  MoveL 5419 to (-31.64, 163.21, 88.06) mm, rotated rx 180 ry 0 rz 180 deg; joints [-52.884, -13.901, 88.099, 78.356, 54.505, -70.46]
  Call Extruder(2.18198)
  MoveL 5420 to (-31.93, 163.09, 88.06) mm, rotated rx 180 ry 0 rz -180 deg; joints [-52.91, -13.939, 88.128, 78.36, 54.532, -70.455]
  MoveL 5421 to (-31.93, 163.09, 88.06) mm, rotated rx 180 ry 0 rz -180 deg; joints [-52.91, -13.939, 88.128, 78.36, 54.532, -70.455]
  Call Extruder(2.36471)
  MoveL 5422 to (-32.22, 162.97, 88.06) mm, rotated rx 180 ry 0 rz 180 deg; joints [-52.936, -13.978, 88.158, 78.364, 54.558, -70.45]
  MoveL 5423 to (-32.22, 162.97, 88.06) mm, rotated rx 180 ry 0 rz 180 deg; joints [-52.936, -13.978, 88.158, 78.364, 54.558, -70.45]
  Call Extruder(2.53513)
  MoveL 5424 to (-32.49, 162.85, 88.06) mm, rotated rx -180 ry 0 rz 180 deg; joints [-52.96, -14.014, 88.185, 78.368, 54.583, -70.445]
  MoveL 5425 to (-32.49, 162.85, 88.06) mm, rotated rx -180 ry 0 rz 180 deg; joints [-52.96, -14.014, 88.185, 78.368, 54.583, -70.445]
  Call Extruder(2.69310)
  MoveL 5426 to (-32.74, 162.74, 88.06) mm, rotated rx 180 ry 0 rz 180 deg; joints [-52.982, -14.048, 88.211, 78.372, 54.605, -70.44]
  MoveL 5427 to (-32.74, 162.74, 88.06) mm, rotated rx 180 ry 0 rz 180 deg; joints [-52.982, -14.048, 88.211, 78.372, 54.605, -70.44]
  Call Extruder(2.85168)
  MoveL 5428 to (-32.99, 162.64, 88.06) mm, rotated rx 180 ry 0 rz -180 deg; joints [-53.004, -14.082, 88.236, 78.375, 54.627, -70.436]
  MoveL 5429 to (-32.99, 162.64, 88.06) mm, rotated rx 180 ry 0 rz -180 deg; joints [-53.004, -14.082, 88.236, 78.375, 54.627, -70.436]
  Call Extruder(3.05785)
  MoveL 5430 to (-33.29, 162.46, 88.06) mm, rotated rx 180 ry 0 rz 180 deg; joints [-53.026, -14.128, 88.271, 78.376, 54.651, -70.428]
  MoveL 5431 to (-33.29, 162.46, 88.06) mm, rotated rx 180 ry 0 rz 180 deg; joints [-53.026, -14.128, 88.271, 78.376, 54.651, -70.428]
  Call Extruder(3.26479)
  MoveL 5432 to (-33.6, 162.29, 88.06) mm, rotated rx 180 ry 0 rz 180 deg; joints [-53.049, -14.174, 88.306, 78.378, 54.674, -70.42]
  MoveL 5433 to (-33.6, 162.29, 88.06) mm, rotated rx 180 ry 0 rz 180 deg; joints [-53.049, -14.174, 88.306, 78.378, 54.674, -70.42]
  Call Extruder(3.47251)
  MoveL 5434 to (-33.9, 162.11, 88.06) mm, rotated rx 180 ry 0 rz 180 deg; joints [-53.071, -14.22, 88.34, 78.379, 54.698, -70.411]
  MoveL 5435 to (-33.9, 162.11, 88.06) mm, rotated rx 180 ry 0 rz 180 deg; joints [-53.071, -14.22, 88.34, 78.379, 54.698, -70.411]
  Call Extruder(3.68102)
  MoveL 5436 to (-34.21, 161.94, 88.06) mm, rotated rx 180 ry 0 rz 180 deg; joints [-53.094, -14.266, 88.375, 78.381, 54.721, -70.403]
  MoveL 5437 to (-34.21, 161.94, 88.06) mm, rotated rx 180 ry 0 rz 180 deg; joints [-53.094, -14.266, 88.375, 78.381, 54.721, -70.403]
  Call Extruder(3.86055)
  MoveL 5438 to (-34.45, 161.76, 88.06) mm, rotated rx 180 ry 0 rz 180 deg; joints [-53.109, -14.307, 88.406, 78.38, 54.737, -70.394]
  MoveL 5439 to (-34.45, 161.76, 88.06) mm, rotated rx 180 ry 0 rz 180 deg; joints [-53.109, -14.307, 88.406, 78.38, 54.737, -70.394]
  Call Extruder(4.19399)
  MoveL 5440 to (-34.9, 161.43, 88.06) mm, rotated rx 180 ry 0 rz 180 deg; joints [-53.135, -14.383, 88.463, 78.378, 54.766, -70.378]
  MoveL 5441 to (-34.9, 161.43, 88.06) mm, rotated rx 180 ry 0 rz 180 deg; joints [-53.135, -14.383, 88.463, 78.378, 54.766, -70.378]
  Call Extruder(4.52861)
  MoveL 5442 to (-35.35, 161.1, 88.06) mm, rotated rx -180 ry 0 rz 180 deg; joints [-53.163, -14.458, 88.52, 78.376, 54.795, -70.362]
  Call Extruder(5.35652)
  MoveL 5443 to (-36.39, 160.19, 88.06) mm, rotated rx 180 ry 0 rz 180 deg; joints [-53.209, -14.651, 88.664, 78.362, 54.849, -70.315]
  Call Extruder(6.18445)
  MoveL 5444 to (-37.3, 159.15, 88.06) mm, rotated rx 180 ry 0 rz -180 deg; joints [-53.227, -14.846, 88.809, 78.335, 54.876, -70.26]
  Call Extruder(6.35176)
  MoveL 5445 to (-37.47, 158.93, 88.06) mm, rotated rx 180 ry 0 rz -180 deg; joints [-53.227, -14.886, 88.839, 78.327, 54.878, -70.247]
  MoveL 5446 to (-37.47, 158.93, 88.06) mm, rotated rx 180 ry 0 rz -180 deg; joints [-53.227, -14.886, 88.839, 78.327, 54.878, -70.247]
  Call Extruder(6.68519)
  MoveL 5447 to (-37.8, 158.48, 88.06) mm, rotated rx -180 ry 0 rz 180 deg; joints [-53.226, -14.965, 88.897, 78.313, 54.881, -70.223]
  MoveL 5448 to (-37.8, 158.48, 88.06) mm, rotated rx -180 ry 0 rz 180 deg; joints [-53.226, -14.965, 88.897, 78.313, 54.881, -70.223]
  Call Extruder(7.01743)
  MoveL 5449 to (-38.12, 158.02, 88.06) mm, rotated rx -180 ry 0 rz 180 deg; joints [-53.224, -15.044, 88.956, 78.298, 54.884, -70.198]
  MoveL 5450 to (-38.12, 158.02, 88.06) mm, rotated rx -180 ry 0 rz 180 deg; joints [-53.224, -15.044, 88.956, 78.298, 54.884, -70.198]
  Call Extruder(7.13510)
  MoveL 5451 to (-38.22, 157.85, 88.06) mm, rotated rx 180 ry 0 rz 180 deg; joints [-53.221, -15.072, 88.977, 78.292, 54.882, -70.188]
  MoveL 5452 to (-38.22, 157.85, 88.06) mm, rotated rx 180 ry 0 rz 180 deg; joints [-53.221, -15.072, 88.977, 78.292, 54.882, -70.188]
  Call Extruder(7.34283)
  MoveL 5453 to (-38.4, 157.55, 88.06) mm, rotated rx -180 ry 0 rz 180 deg; joints [-53.214, -15.121, 89.013, 78.28, 54.878, -70.171]
  MoveL 5454 to (-38.4, 157.55, 88.06) mm, rotated rx -180 ry 0 rz 180 deg; joints [-53.214, -15.121, 89.013, 78.28, 54.878, -70.171]
  Call Extruder(7.54978)
  MoveL 5455 to (-38.57, 157.25, 88.06) mm, rotated rx 180 ry 0 rz 180 deg; joints [-53.207, -15.171, 89.05, 78.268, 54.874, -70.154]
  MoveL 5456 to (-38.57, 157.25, 88.06) mm, rotated rx 180 ry 0 rz 180 deg; joints [-53.207, -15.171, 89.05, 78.268, 54.874, -70.154]
  Call Extruder(7.75595)
  MoveL 5457 to (-38.75, 156.94, 88.06) mm, rotated rx -180 ry 0 rz 180 deg; joints [-53.2, -15.22, 89.086, 78.256, 54.87, -70.137]
  MoveL 5458 to (-38.75, 156.94, 88.06) mm, rotated rx -180 ry 0 rz 180 deg; joints [-53.2, -15.22, 89.086, 78.256, 54.87, -70.137]
  Call Extruder(7.93763)
  MoveL 5459 to (-38.89, 156.66, 88.06) mm, rotated rx -180 ry 0 rz 180 deg; joints [-53.191, -15.263, 89.118, 78.245, 54.864, -70.121]
  MoveL 5460 to (-38.89, 156.66, 88.06) mm, rotated rx -180 ry 0 rz 180 deg; joints [-53.191, -15.263, 89.118, 78.245, 54.864, -70.121]
  Call Extruder(8.09561)
  MoveL 5461 to (-39, 156.42, 88.06) mm, rotated rx -180 ry 0 rz 180 deg; joints [-53.18, -15.301, 89.145, 78.234, 54.856, -70.107]
  MoveL 5462 to (-39, 156.42, 88.06) mm, rotated rx -180 ry 0 rz 180 deg; joints [-53.18, -15.301, 89.145, 78.234, 54.856, -70.107]
  Call Extruder(8.25300)
  MoveL 5463 to (-39.11, 156.17, 88.06) mm, rotated rx -180 ry 0 rz 180 deg; joints [-53.17, -15.338, 89.173, 78.222, 54.848, -70.092]
  MoveL 5464 to (-39.11, 156.17, 88.06) mm, rotated rx -180 ry 0 rz 180 deg; joints [-53.17, -15.338, 89.173, 78.222, 54.848, -70.092]
  Call Extruder(8.43571)
  MoveL 5465 to (-39.22, 155.88, 88.06) mm, rotated rx 180 ry 0 rz 180 deg; joints [-53.156, -15.381, 89.205, 78.209, 54.838, -70.075]
  MoveL 5466 to (-39.22, 155.88, 88.06) mm, rotated rx 180 ry 0 rz 180 deg; joints [-53.156, -15.381, 89.205, 78.209, 54.838, -70.075]
  Call Extruder(8.61768)
  MoveL 5467 to (-39.35, 155.58, 88.06) mm, rotated rx 180 ry 0 rz 180 deg; joints [-53.143, -15.425, 89.236, 78.195, 54.828, -70.058]
  MoveL 5468 to (-39.35, 155.58, 88.06) mm, rotated rx 180 ry 0 rz 180 deg; joints [-53.143, -15.425, 89.236, 78.195, 54.828, -70.058]
  Call Extruder(8.76501)
  MoveL 5469 to (-39.44, 155.34, 88.06) mm, rotated rx 180 ry 0 rz 180 deg; joints [-53.131, -15.459, 89.262, 78.184, 54.819, -70.044]
  MoveL 5470 to (-39.44, 155.34, 88.06) mm, rotated rx 180 ry 0 rz 180 deg; joints [-53.131, -15.459, 89.262, 78.184, 54.819, -70.044]
  Call Extruder(8.87824)
  MoveL 5471 to (-39.5, 155.15, 88.06) mm, rotated rx -180 ry 0 rz 180 deg; joints [-53.121, -15.486, 89.281, 78.175, 54.81, -70.033]
  MoveL 5472 to (-39.5, 155.15, 88.06) mm, rotated rx -180 ry 0 rz 180 deg; joints [-53.121, -15.486, 89.281, 78.175, 54.81, -70.033]
  Call Extruder(8.99103)
  MoveL 5473 to (-39.56, 154.97, 88.06) mm, rotated rx 180 ry 0 rz 180 deg; joints [-53.11, -15.513, 89.301, 78.165, 54.801, -70.022]
  MoveL 5474 to (-39.56, 154.97, 88.06) mm, rotated rx 180 ry 0 rz 180 deg; joints [-53.11, -15.513, 89.301, 78.165, 54.801, -70.022]
  Call Extruder(9.10338)
  MoveL 5475 to (-39.62, 154.78, 88.06) mm, rotated rx 180 ry 0 rz 180 deg; joints [-53.099, -15.539, 89.32, 78.156, 54.793, -70.011]
  MoveL 5476 to (-39.62, 154.78, 88.06) mm, rotated rx 180 ry 0 rz 180 deg; joints [-53.099, -15.539, 89.32, 78.156, 54.793, -70.011]
  Call Extruder(9.21528)
  MoveL 5477 to (-39.68, 154.59, 88.06) mm, rotated rx 180 ry 0 rz 180 deg; joints [-53.088, -15.566, 89.34, 78.146, 54.784, -70]
  MoveL 5478 to (-39.68, 154.59, 88.06) mm, rotated rx 180 ry 0 rz 180 deg; joints [-53.088, -15.566, 89.34, 78.146, 54.784, -70]
  Call Extruder(9.33668)
  MoveL 5479 to (-39.75, 154.38, 88.06) mm, rotated rx -180 ry 0 rz 180 deg; joints [-53.076, -15.594, 89.361, 78.136, 54.774, -69.988]
  MoveL 5480 to (-39.75, 154.38, 88.06) mm, rotated rx -180 ry 0 rz 180 deg; joints [-53.076, -15.594, 89.361, 78.136, 54.774, -69.988]
  Call Extruder(9.46747)
  MoveL 5481 to (-39.81, 154.16, 88.06) mm, rotated rx 180 ry 0 rz 180 deg; joints [-53.063, -15.625, 89.383, 78.124, 54.763, -69.974]
  MoveL 5482 to (-39.81, 154.16, 88.06) mm, rotated rx 180 ry 0 rz 180 deg; joints [-53.063, -15.625, 89.383, 78.124, 54.763, -69.974]
  Call Extruder(9.59770)
  MoveL 5483 to (-39.88, 153.94, 88.06) mm, rotated rx 180 ry 0 rz 180 deg; joints [-53.049, -15.656, 89.406, 78.113, 54.752, -69.961]
  MoveL 5484 to (-39.88, 153.94, 88.06) mm, rotated rx 180 ry 0 rz 180 deg; joints [-53.049, -15.656, 89.406, 78.113, 54.752, -69.961]
  Call Extruder(9.72737)
  MoveL 5485 to (-39.95, 153.71, 88.06) mm, rotated rx 180 ry 0 rz 180 deg; joints [-53.036, -15.687, 89.428, 78.102, 54.741, -69.948]
  MoveL 5486 to (-39.95, 153.71, 88.06) mm, rotated rx 180 ry 0 rz 180 deg; joints [-53.036, -15.687, 89.428, 78.102, 54.741, -69.948]
  Call Extruder(9.85647)
  MoveL 5487 to (-40.02, 153.49, 88.06) mm, rotated rx 180 ry 0 rz 180 deg; joints [-53.022, -15.718, 89.451, 78.09, 54.73, -69.934]
  MoveL 5488 to (-40.02, 153.49, 88.06) mm, rotated rx 180 ry 0 rz 180 deg; joints [-53.022, -15.718, 89.451, 78.09, 54.73, -69.934]
  Call Extruder(9.97156)
  MoveL 5489 to (-40.06, 153.28, 88.06) mm, rotated rx -180 ry 0 rz 180 deg; joints [-53.007, -15.745, 89.471, 78.079, 54.718, -69.922]
  MoveL 5490 to (-40.06, 153.28, 88.06) mm, rotated rx -180 ry 0 rz 180 deg; joints [-53.007, -15.745, 89.471, 78.079, 54.718, -69.922]
  Call Extruder(10.08619)
  MoveL 5491 to (-40.11, 153.08, 88.06) mm, rotated rx 180 ry 0 rz 180 deg; joints [-52.993, -15.772, 89.49, 78.067, 54.706, -69.91]
  MoveL 5492 to (-40.11, 153.08, 88.06) mm, rotated rx 180 ry 0 rz 180 deg; joints [-52.993, -15.772, 89.49, 78.067, 54.706, -69.91]
  Call Extruder(10.20038)
  MoveL 5493 to (-40.15, 152.88, 88.06) mm, rotated rx 180 ry 0 rz 180 deg; joints [-52.978, -15.799, 89.509, 78.056, 54.693, -69.897]
  MoveL 5494 to (-40.15, 152.88, 88.06) mm, rotated rx 180 ry 0 rz 180 deg; joints [-52.978, -15.799, 89.509, 78.056, 54.693, -69.897]
  Call Extruder(10.31411)
  MoveL 5495 to (-40.2, 152.67, 88.06) mm, rotated rx 180 ry 0 rz 180 deg; joints [-52.963, -15.826, 89.529, 78.045, 54.681, -69.885]
  MoveL 5496 to (-40.2, 152.67, 88.06) mm, rotated rx 180 ry 0 rz 180 deg; joints [-52.963, -15.826, 89.529, 78.045, 54.681, -69.885]
  Call Extruder(10.43953)
  MoveL 5497 to (-40.24, 152.45, 88.06) mm, rotated rx 180 ry 0 rz 180 deg; joints [-52.946, -15.855, 89.55, 78.032, 54.667, -69.871]
  MoveL 5498 to (-40.24, 152.45, 88.06) mm, rotated rx 180 ry 0 rz 180 deg; joints [-52.946, -15.855, 89.55, 78.032, 54.667, -69.871]
  Call Extruder(10.57651)
  MoveL 5499 to (-40.29, 152.2, 88.06) mm, rotated rx 180 ry 0 rz 180 deg; joints [-52.928, -15.887, 89.574, 78.018, 54.651, -69.856]
  MoveL 5500 to (-40.29, 152.2, 88.06) mm, rotated rx 180 ry 0 rz 180 deg; joints [-52.928, -15.887, 89.574, 78.018, 54.651, -69.856]
  Call Extruder(10.71287)
  MoveL 5501 to (-40.34, 151.95, 88.06) mm, rotated rx -180 ry 0 rz 180 deg; joints [-52.909, -15.92, 89.597, 78.004, 54.635, -69.841]
  MoveL 5502 to (-40.34, 151.95, 88.06) mm, rotated rx -180 ry 0 rz 180 deg; joints [-52.909, -15.92, 89.597, 78.004, 54.635, -69.841]
  Call Extruder(10.84863)
  MoveL 5503 to (-40.39, 151.7, 88.06) mm, rotated rx 180 ry 0 rz -180 deg; joints [-52.89, -15.952, 89.621, 77.99, 54.62, -69.825]
  MoveL 5504 to (-40.39, 151.7, 88.06) mm, rotated rx 180 ry 0 rz -180 deg; joints [-52.89, -15.952, 89.621, 77.99, 54.62, -69.825]
  Call Extruder(10.98377)
  MoveL 5505 to (-40.44, 151.45, 88.06) mm, rotated rx 180 ry 0 rz -180 deg; joints [-52.871, -15.984, 89.644, 77.976, 54.604, -69.81]
  MoveL 5506 to (-40.44, 151.45, 88.06) mm, rotated rx 180 ry 0 rz -180 deg; joints [-52.871, -15.984, 89.644, 77.976, 54.604, -69.81]
  Call Extruder(11.11831)
  MoveL 5507 to (-40.49, 151.2, 88.06) mm, rotated rx -180 ry 0 rz 180 deg; joints [-52.853, -16.016, 89.667, 77.962, 54.588, -69.795]
  MoveL 5508 to (-40.49, 151.2, 88.06) mm, rotated rx -180 ry 0 rz 180 deg; joints [-52.853, -16.016, 89.667, 77.962, 54.588, -69.795]
  Call Extruder(11.25223)
  MoveL 5509 to (-40.54, 150.95, 88.06) mm, rotated rx -180 ry 0 rz 180 deg; joints [-52.834, -16.048, 89.69, 77.947, 54.572, -69.779]
  MoveL 5510 to (-40.54, 150.95, 88.06) mm, rotated rx -180 ry 0 rz 180 deg; joints [-52.834, -16.048, 89.69, 77.947, 54.572, -69.779]
  Call Extruder(11.40009)
  MoveL 5511 to (-40.59, 150.67, 88.06) mm, rotated rx 180 ry 0 rz 180 deg; joints [-52.812, -16.084, 89.716, 77.931, 54.554, -69.762]
  MoveL 5512 to (-40.59, 150.67, 88.06) mm, rotated rx 180 ry 0 rz 180 deg; joints [-52.812, -16.084, 89.716, 77.931, 54.554, -69.762]
  Call Extruder(11.56181)
  MoveL 5513 to (-40.64, 150.37, 88.06) mm, rotated rx 180 ry 0 rz 180 deg; joints [-52.787, -16.122, 89.744, 77.913, 54.533, -69.743]
  MoveL 5514 to (-40.64, 150.37, 88.06) mm, rotated rx 180 ry 0 rz 180 deg; joints [-52.787, -16.122, 89.744, 77.913, 54.533, -69.743]
  Call Extruder(11.72281)
  MoveL 5515 to (-40.69, 150.06, 88.06) mm, rotated rx 180 ry 0 rz 180 deg; joints [-52.762, -16.161, 89.771, 77.895, 54.512, -69.724]
  MoveL 5516 to (-40.69, 150.06, 88.06) mm, rotated rx 180 ry 0 rz 180 deg; joints [-52.762, -16.161, 89.771, 77.895, 54.512, -69.724]
  Call Extruder(11.88308)
  MoveL 5517 to (-40.73, 149.76, 88.06) mm, rotated rx 180 ry 0 rz 180 deg; joints [-52.737, -16.199, 89.799, 77.877, 54.491, -69.705]
  MoveL 5518 to (-40.73, 149.76, 88.06) mm, rotated rx 180 ry 0 rz 180 deg; joints [-52.737, -16.199, 89.799, 77.877, 54.491, -69.705]
  Call Extruder(12.04262)
  MoveL 5519 to (-40.78, 149.45, 88.06) mm, rotated rx -180 ry 0 rz -180 deg; joints [-52.712, -16.237, 89.827, 77.859, 54.469, -69.686]
  MoveL 5520 to (-40.78, 149.45, 88.06) mm, rotated rx -180 ry 0 rz -180 deg; joints [-52.712, -16.237, 89.827, 77.859, 54.469, -69.686]
  Call Extruder(12.20144)
  MoveL 5521 to (-40.83, 149.14, 88.06) mm, rotated rx -180 ry 0 rz -180 deg; joints [-52.687, -16.276, 89.854, 77.841, 54.448, -69.667]
  MoveL 5522 to (-40.83, 149.14, 88.06) mm, rotated rx -180 ry 0 rz -180 deg; joints [-52.687, -16.276, 89.854, 77.841, 54.448, -69.667]
  Call Extruder(12.38010)
  MoveL 5523 to (-40.88, 148.8, 88.06) mm, rotated rx 180 ry 0 rz 180 deg; joints [-52.658, -16.319, 89.885, 77.82, 54.423, -69.645]
  MoveL 5524 to (-40.88, 148.8, 88.06) mm, rotated rx 180 ry 0 rz 180 deg; joints [-52.658, -16.319, 89.885, 77.82, 54.423, -69.645]
  Call Extruder(12.57854)
  MoveL 5525 to (-40.93, 148.41, 88.06) mm, rotated rx 180 ry 0 rz 180 deg; joints [-52.624, -16.366, 89.919, 77.796, 54.394, -69.62]
  MoveL 5526 to (-40.93, 148.41, 88.06) mm, rotated rx 180 ry 0 rz 180 deg; joints [-52.624, -16.366, 89.919, 77.796, 54.394, -69.62]
  Call Extruder(12.77611)
  MoveL 5527 to (-40.97, 148.02, 88.06) mm, rotated rx 180 ry 0 rz 180 deg; joints [-52.59, -16.413, 89.953, 77.772, 54.365, -69.596]
  MoveL 5528 to (-40.97, 148.02, 88.06) mm, rotated rx 180 ry 0 rz 180 deg; joints [-52.59, -16.413, 89.953, 77.772, 54.365, -69.596]
  Call Extruder(12.97282)
  MoveL 5529 to (-41.02, 147.63, 88.06) mm, rotated rx 180 ry 0 rz 180 deg; joints [-52.556, -16.46, 89.986, 77.748, 54.336, -69.571]
  MoveL 5530 to (-41.02, 147.63, 88.06) mm, rotated rx 180 ry 0 rz 180 deg; joints [-52.556, -16.46, 89.986, 77.748, 54.336, -69.571]
  Call Extruder(13.16866)
  MoveL 5531 to (-41.06, 147.25, 88.06) mm, rotated rx 180 ry 0 rz 180 deg; joints [-52.521, -16.508, 90.02, 77.724, 54.307, -69.546]
  MoveL 5532 to (-41.06, 147.25, 88.06) mm, rotated rx 180 ry 0 rz 180 deg; joints [-52.521, -16.508, 90.02, 77.724, 54.307, -69.546]
  Call Extruder(13.46406)
  MoveL 5533 to (-41.11, 146.66, 88.06) mm, rotated rx 180 ry 0 rz 180 deg; joints [-52.466, -16.577, 90.07, 77.686, 54.259, -69.508]
  MoveL 5534 to (-41.11, 146.66, 88.06) mm, rotated rx 180 ry 0 rz 180 deg; joints [-52.466, -16.577, 90.07, 77.686, 54.259, -69.508]
  Call Extruder(13.75812)
  MoveL 5535 to (-41.15, 146.07, 88.06) mm, rotated rx -180 ry 0 rz 180 deg; joints [-52.411, -16.647, 90.119, 77.648, 54.212, -69.47]
  MoveL 5536 to (-41.15, 146.07, 88.06) mm, rotated rx -180 ry 0 rz 180 deg; joints [-52.411, -16.647, 90.119, 77.648, 54.212, -69.47]
  Call Extruder(14.05085)
  MoveL 5537 to (-41.2, 145.48, 88.06) mm, rotated rx -180 ry 0 rz 180 deg; joints [-52.355, -16.717, 90.169, 77.61, 54.164, -69.432]
  MoveL 5538 to (-41.2, 145.48, 88.06) mm, rotated rx -180 ry 0 rz 180 deg; joints [-52.355, -16.717, 90.169, 77.61, 54.164, -69.432]
  Call Extruder(14.62431)
  MoveL 5539 to (-41.25, 144.32, 88.06) mm, rotated rx 180 ry 0 rz 180 deg; joints [-52.239, -16.85, 90.263, 77.532, 54.063, -69.356]
  MoveL 5540 to (-41.25, 144.32, 88.06) mm, rotated rx 180 ry 0 rz 180 deg; joints [-52.239, -16.85, 90.263, 77.532, 54.063, -69.356]
  Call Extruder(15.33827)
  MoveL 5541 to (-41.29, 142.86, 88.06) mm, rotated rx 180 ry 0 rz 180 deg; joints [-52.09, -17.014, 90.38, 77.432, 53.934, -69.259]
  Call Extruder(57.40309)
  MoveL 5542 to (-41.29, 57.14, 88.06) mm, rotated rx 180 ry 0 rz 180 deg; joints [-40.759, -25.558, 95.751, 68.538, 44.549, -61.117]
  Call Extruder(57.83165)
  MoveL 5543 to (-41.27, 56.26, 88.06) mm, rotated rx -180 ry 0 rz -180 deg; joints [-40.614, -25.632, 95.792, 68.407, 44.435, -61.001]
  MoveL 5544 to (-41.27, 56.26, 88.06) mm, rotated rx -180 ry 0 rz -180 deg; joints [-40.614, -25.632, 95.792, 68.407, 44.435, -61.001]
  Call Extruder(58.40510)
  MoveL 5545 to (-41.23, 55.1, 88.06) mm, rotated rx 180 ry 0 rz -180 deg; joints [-40.419, -25.728, 95.844, 68.23, 44.28, -60.846]
  MoveL 5546 to (-41.23, 55.1, 88.06) mm, rotated rx 180 ry 0 rz -180 deg; joints [-40.419, -25.728, 95.844, 68.23, 44.28, -60.846]
  Call Extruder(58.83942)
  MoveL 5547 to (-41.18, 54.23, 88.06) mm, rotated rx 180 ry 0 rz 180 deg; joints [-40.269, -25.799, 95.883, 68.094, 44.161, -60.728]
  MoveL 5548 to (-41.18, 54.23, 88.06) mm, rotated rx 180 ry 0 rz 180 deg; joints [-40.269, -25.799, 95.883, 68.094, 44.161, -60.728]
  Call Extruder(59.13348)
  MoveL 5549 to (-41.13, 53.64, 88.06) mm, rotated rx 180 ry 0 rz 180 deg; joints [-40.165, -25.845, 95.908, 68.001, 44.078, -60.648]
  MoveL 5550 to (-41.13, 53.64, 88.06) mm, rotated rx 180 ry 0 rz 180 deg; joints [-40.165, -25.845, 95.908, 68.001, 44.078, -60.648]
  Call Extruder(59.42888)
  MoveL 5551 to (-41.09, 53.05, 88.06) mm, rotated rx 180 ry 0 rz 180 deg; joints [-40.062, -25.891, 95.933, 67.908, 43.996, -60.568]
  MoveL 5552 to (-41.09, 53.05, 88.06) mm, rotated rx 180 ry 0 rz 180 deg; joints [-40.062, -25.891, 95.933, 67.908, 43.996, -60.568]
  Call Extruder(59.67512)
  MoveL 5553 to (-41.04, 52.56, 88.06) mm, rotated rx 180 ry 0 rz 180 deg; joints [-39.975, -25.928, 95.953, 67.83, 43.927, -60.501]
  MoveL 5554 to (-41.04, 52.56, 88.06) mm, rotated rx 180 ry 0 rz 180 deg; joints [-39.975, -25.928, 95.953, 67.83, 43.927, -60.501]
  Call Extruder(59.87182)
  MoveL 5555 to (-40.99, 52.17, 88.06) mm, rotated rx -180 ry 0 rz 180 deg; joints [-39.904, -25.957, 95.969, 67.768, 43.87, -60.447]
  MoveL 5556 to (-40.99, 52.17, 88.06) mm, rotated rx -180 ry 0 rz 180 deg; joints [-39.904, -25.957, 95.969, 67.768, 43.87, -60.447]
  Call Extruder(60.06940)
  MoveL 5557 to (-40.95, 51.78, 88.06) mm, rotated rx 180 ry 0 rz 180 deg; joints [-39.833, -25.985, 95.984, 67.705, 43.814, -60.394]
  MoveL 5558 to (-40.95, 51.78, 88.06) mm, rotated rx 180 ry 0 rz 180 deg; joints [-39.833, -25.985, 95.984, 67.705, 43.814, -60.394]
  Call Extruder(60.26784)
  MoveL 5559 to (-40.9, 51.4, 88.06) mm, rotated rx -180 ry 0 rz -180 deg; joints [-39.763, -26.013, 96, 67.642, 43.757, -60.34]
  MoveL 5560 to (-40.9, 51.4, 88.06) mm, rotated rx -180 ry 0 rz -180 deg; joints [-39.763, -26.013, 96, 67.642, 43.757, -60.34]
  Call Extruder(60.46715)
  MoveL 5561 to (-40.86, 51.01, 88.06) mm, rotated rx 180 ry 0 rz 180 deg; joints [-39.692, -26.042, 96.015, 67.578, 43.7, -60.286]
  MoveL 5562 to (-40.86, 51.01, 88.06) mm, rotated rx 180 ry 0 rz 180 deg; joints [-39.692, -26.042, 96.015, 67.578, 43.7, -60.286]
  Call Extruder(60.62596)
  MoveL 5563 to (-40.81, 50.7, 88.06) mm, rotated rx -180 ry 0 rz -180 deg; joints [-39.634, -26.063, 96.026, 67.528, 43.654, -60.243]
  MoveL 5564 to (-40.81, 50.7, 88.06) mm, rotated rx -180 ry 0 rz -180 deg; joints [-39.634, -26.063, 96.026, 67.528, 43.654, -60.243]
  Call Extruder(60.78551)
  MoveL 5565 to (-40.76, 50.4, 88.06) mm, rotated rx 180 ry 0 rz -180 deg; joints [-39.576, -26.084, 96.038, 67.477, 43.607, -60.2]
  MoveL 5566 to (-40.76, 50.4, 88.06) mm, rotated rx 180 ry 0 rz -180 deg; joints [-39.576, -26.084, 96.038, 67.477, 43.607, -60.2]
  Call Extruder(60.94578)
  MoveL 5567 to (-40.71, 50.09, 88.06) mm, rotated rx 180 ry 0 rz -180 deg; joints [-39.518, -26.104, 96.049, 67.426, 43.561, -60.157]
  MoveL 5568 to (-40.71, 50.09, 88.06) mm, rotated rx 180 ry 0 rz -180 deg; joints [-39.518, -26.104, 96.049, 67.426, 43.561, -60.157]
  Call Extruder(61.10677)
  MoveL 5569 to (-40.66, 49.79, 88.06) mm, rotated rx 180 ry 0 rz 180 deg; joints [-39.46, -26.125, 96.06, 67.374, 43.514, -60.114]
  MoveL 5570 to (-40.66, 49.79, 88.06) mm, rotated rx 180 ry 0 rz 180 deg; joints [-39.46, -26.125, 96.06, 67.374, 43.514, -60.114]
  Call Extruder(61.26850)
  MoveL 5571 to (-40.61, 49.48, 88.06) mm, rotated rx -180 ry 0 rz 180 deg; joints [-39.402, -26.146, 96.072, 67.323, 43.468, -60.07]
  MoveL 5572 to (-40.61, 49.48, 88.06) mm, rotated rx -180 ry 0 rz 180 deg; joints [-39.402, -26.146, 96.072, 67.323, 43.468, -60.07]
  Call Extruder(61.43095)
  MoveL 5573 to (-40.57, 49.17, 88.06) mm, rotated rx 180 ry 0 rz 180 deg; joints [-39.344, -26.167, 96.083, 67.272, 43.421, -60.027]
  MoveL 5574 to (-40.57, 49.17, 88.06) mm, rotated rx 180 ry 0 rz 180 deg; joints [-39.344, -26.167, 96.083, 67.272, 43.421, -60.027]
  Call Extruder(61.56488)
  MoveL 5575 to (-40.52, 48.93, 88.06) mm, rotated rx 180 ry 0 rz 180 deg; joints [-39.296, -26.183, 96.092, 67.229, 43.382, -59.991]
  MoveL 5576 to (-40.52, 48.93, 88.06) mm, rotated rx 180 ry 0 rz 180 deg; joints [-39.296, -26.183, 96.092, 67.229, 43.382, -59.991]
  Call Extruder(61.69941)
  MoveL 5577 to (-40.47, 48.68, 88.06) mm, rotated rx -180 ry 0 rz 180 deg; joints [-39.247, -26.199, 96.1, 67.186, 43.342, -59.955]
  MoveL 5578 to (-40.47, 48.68, 88.06) mm, rotated rx -180 ry 0 rz 180 deg; joints [-39.247, -26.199, 96.1, 67.186, 43.342, -59.955]
  Call Extruder(61.83456)
  MoveL 5579 to (-40.42, 48.43, 88.06) mm, rotated rx 180 ry 0 rz 180 deg; joints [-39.198, -26.215, 96.109, 67.143, 43.303, -59.92]
  MoveL 5580 to (-40.42, 48.43, 88.06) mm, rotated rx 180 ry 0 rz 180 deg; joints [-39.198, -26.215, 96.109, 67.143, 43.303, -59.92]
  Call Extruder(61.97031)
  MoveL 5581 to (-40.37, 48.18, 88.06) mm, rotated rx -180 ry 0 rz 180 deg; joints [-39.149, -26.231, 96.117, 67.101, 43.263, -59.884]
  MoveL 5582 to (-40.37, 48.18, 88.06) mm, rotated rx -180 ry 0 rz 180 deg; joints [-39.149, -26.231, 96.117, 67.101, 43.263, -59.884]
  Call Extruder(62.10668)
  MoveL 5583 to (-40.32, 47.93, 88.06) mm, rotated rx -180 ry 0 rz 180 deg; joints [-39.1, -26.246, 96.126, 67.058, 43.224, -59.848]
  MoveL 5584 to (-40.32, 47.93, 88.06) mm, rotated rx -180 ry 0 rz 180 deg; joints [-39.1, -26.246, 96.126, 67.058, 43.224, -59.848]
  Call Extruder(62.24365)
  MoveL 5585 to (-40.27, 47.68, 88.06) mm, rotated rx 180 ry 0 rz 180 deg; joints [-39.051, -26.262, 96.134, 67.015, 43.185, -59.812]
  MoveL 5586 to (-40.27, 47.68, 88.06) mm, rotated rx 180 ry 0 rz 180 deg; joints [-39.051, -26.262, 96.134, 67.015, 43.185, -59.812]
  Call Extruder(62.38124)
  MoveL 5587 to (-40.22, 47.43, 88.06) mm, rotated rx 180 ry 0 rz 180 deg; joints [-39.002, -26.278, 96.142, 66.971, 43.145, -59.776]
  MoveL 5588 to (-40.22, 47.43, 88.06) mm, rotated rx 180 ry 0 rz 180 deg; joints [-39.002, -26.278, 96.142, 66.971, 43.145, -59.776]
  Call Extruder(62.49497)
  MoveL 5589 to (-40.17, 47.23, 88.06) mm, rotated rx -180 ry 0 rz 180 deg; joints [-38.962, -26.29, 96.149, 66.936, 43.112, -59.746]
  MoveL 5590 to (-40.17, 47.23, 88.06) mm, rotated rx -180 ry 0 rz 180 deg; joints [-38.962, -26.29, 96.149, 66.936, 43.112, -59.746]
  Call Extruder(62.60915)
  MoveL 5591 to (-40.13, 47.02, 88.06) mm, rotated rx -180 ry 0 rz 180 deg; joints [-38.921, -26.303, 96.156, 66.9, 43.079, -59.716]
  MoveL 5592 to (-40.13, 47.02, 88.06) mm, rotated rx -180 ry 0 rz 180 deg; joints [-38.921, -26.303, 96.156, 66.9, 43.079, -59.716]
  Call Extruder(62.72378)
  MoveL 5593 to (-40.08, 46.82, 88.06) mm, rotated rx -180 ry 0 rz 180 deg; joints [-38.88, -26.315, 96.163, 66.864, 43.046, -59.687]
  MoveL 5594 to (-40.08, 46.82, 88.06) mm, rotated rx -180 ry 0 rz 180 deg; joints [-38.88, -26.315, 96.163, 66.864, 43.046, -59.687]
  Call Extruder(62.83887)
  MoveL 5595 to (-40.04, 46.61, 88.06) mm, rotated rx -180 ry 0 rz 180 deg; joints [-38.839, -26.328, 96.169, 66.828, 43.013, -59.657]
  MoveL 5596 to (-40.04, 46.61, 88.06) mm, rotated rx -180 ry 0 rz 180 deg; joints [-38.839, -26.328, 96.169, 66.828, 43.013, -59.657]
  Call Extruder(62.96111)
  MoveL 5597 to (-39.98, 46.4, 88.06) mm, rotated rx 180 ry 0 rz 180 deg; joints [-38.795, -26.34, 96.176, 66.79, 42.977, -59.625]
  MoveL 5598 to (-39.98, 46.4, 88.06) mm, rotated rx 180 ry 0 rz 180 deg; joints [-38.795, -26.34, 96.176, 66.79, 42.977, -59.625]
  Call Extruder(63.09077)
  MoveL 5599 to (-39.92, 46.18, 88.06) mm, rotated rx 180 ry 0 rz 180 deg; joints [-38.748, -26.351, 96.182, 66.75, 42.938, -59.592]
  MoveL 5600 to (-39.92, 46.18, 88.06) mm, rotated rx 180 ry 0 rz 180 deg; joints [-38.748, -26.351, 96.182, 66.75, 42.938, -59.592]
  Call Extruder(63.22100)
  MoveL 5601 to (-39.85, 45.95, 88.06) mm, rotated rx 180 ry 0 rz 180 deg; joints [-38.7, -26.363, 96.188, 66.709, 42.9, -59.559]
  MoveL 5602 to (-39.85, 45.95, 88.06) mm, rotated rx 180 ry 0 rz 180 deg; joints [-38.7, -26.363, 96.188, 66.709, 42.9, -59.559]
  Call Extruder(63.35179)
  MoveL 5603 to (-39.78, 45.73, 88.06) mm, rotated rx 180 ry 0 rz 180 deg; joints [-38.653, -26.374, 96.194, 66.668, 42.861, -59.526]
  MoveL 5604 to (-39.78, 45.73, 88.06) mm, rotated rx 180 ry 0 rz 180 deg; joints [-38.653, -26.374, 96.194, 66.668, 42.861, -59.526]
  Call Extruder(63.48315)
  MoveL 5605 to (-39.71, 45.51, 88.06) mm, rotated rx -180 ry 0 rz 180 deg; joints [-38.605, -26.386, 96.2, 66.628, 42.822, -59.493]
  MoveL 5606 to (-39.71, 45.51, 88.06) mm, rotated rx -180 ry 0 rz 180 deg; joints [-38.605, -26.386, 96.2, 66.628, 42.822, -59.493]
  Call Extruder(63.59505)
  MoveL 5607 to (-39.65, 45.32, 88.06) mm, rotated rx 180 ry 0 rz 180 deg; joints [-38.565, -26.395, 96.205, 66.593, 42.789, -59.465]
  MoveL 5608 to (-39.65, 45.32, 88.06) mm, rotated rx 180 ry 0 rz 180 deg; joints [-38.565, -26.395, 96.205, 66.593, 42.789, -59.465]
  Call Extruder(63.70740)
  MoveL 5609 to (-39.59, 45.13, 88.06) mm, rotated rx 180 ry 0 rz 180 deg; joints [-38.524, -26.404, 96.21, 66.558, 42.756, -59.437]
  MoveL 5610 to (-39.59, 45.13, 88.06) mm, rotated rx 180 ry 0 rz 180 deg; joints [-38.524, -26.404, 96.21, 66.558, 42.756, -59.437]
  Call Extruder(63.82019)
  MoveL 5611 to (-39.53, 44.94, 88.06) mm, rotated rx 180 ry 0 rz 180 deg; joints [-38.483, -26.414, 96.215, 66.524, 42.722, -59.409]
  MoveL 5612 to (-39.53, 44.94, 88.06) mm, rotated rx 180 ry 0 rz 180 deg; joints [-38.483, -26.414, 96.215, 66.524, 42.722, -59.409]
  Call Extruder(63.93342)
  MoveL 5613 to (-39.47, 44.75, 88.06) mm, rotated rx 180 ry 0 rz 180 deg; joints [-38.443, -26.423, 96.22, 66.489, 42.689, -59.38]
  MoveL 5614 to (-39.47, 44.75, 88.06) mm, rotated rx 180 ry 0 rz 180 deg; joints [-38.443, -26.423, 96.22, 66.489, 42.689, -59.38]
  Call Extruder(64.04710)
  MoveL 5615 to (-39.41, 44.56, 88.06) mm, rotated rx -180 ry 0 rz 180 deg; joints [-38.402, -26.432, 96.225, 66.454, 42.656, -59.352]
  MoveL 5616 to (-39.41, 44.56, 88.06) mm, rotated rx -180 ry 0 rz 180 deg; joints [-38.402, -26.432, 96.225, 66.454, 42.656, -59.352]
  Call Extruder(64.22906)
  MoveL 5617 to (-39.29, 44.27, 88.06) mm, rotated rx -180 ry 0 rz 180 deg; joints [-38.335, -26.443, 96.231, 66.399, 42.601, -59.308]
  MoveL 5618 to (-39.29, 44.27, 88.06) mm, rotated rx -180 ry 0 rz 180 deg; joints [-38.335, -26.443, 96.231, 66.399, 42.601, -59.308]
  Call Extruder(64.41178)
  MoveL 5619 to (-39.17, 43.98, 88.06) mm, rotated rx 180 ry 0 rz 180 deg; joints [-38.269, -26.455, 96.237, 66.343, 42.545, -59.264]
  MoveL 5620 to (-39.17, 43.98, 88.06) mm, rotated rx 180 ry 0 rz 180 deg; joints [-38.269, -26.455, 96.237, 66.343, 42.545, -59.264]
  Call Extruder(64.58219)
  MoveL 5621 to (-39.05, 43.71, 88.06) mm, rotated rx 180 ry 0 rz 180 deg; joints [-38.207, -26.465, 96.243, 66.291, 42.494, -59.223]
  MoveL 5622 to (-39.05, 43.71, 88.06) mm, rotated rx 180 ry 0 rz 180 deg; joints [-38.207, -26.465, 96.243, 66.291, 42.494, -59.223]
  Call Extruder(64.74018)
  MoveL 5623 to (-38.94, 43.46, 88.06) mm, rotated rx 180 ry 0 rz 180 deg; joints [-38.149, -26.474, 96.248, 66.243, 42.447, -59.185]
  MoveL 5624 to (-38.94, 43.46, 88.06) mm, rotated rx 180 ry 0 rz 180 deg; joints [-38.149, -26.474, 96.248, 66.243, 42.447, -59.185]
  Call Extruder(64.89877)
  MoveL 5625 to (-38.84, 43.21, 88.06) mm, rotated rx 180 ry 0 rz 180 deg; joints [-38.092, -26.484, 96.253, 66.195, 42.399, -59.146]
  MoveL 5626 to (-38.84, 43.21, 88.06) mm, rotated rx 180 ry 0 rz 180 deg; joints [-38.092, -26.484, 96.253, 66.195, 42.399, -59.146]
  Call Extruder(65.10493)
  MoveL 5627 to (-38.66, 42.91, 88.06) mm, rotated rx 180 ry 0 rz 180 deg; joints [-38.016, -26.49, 96.256, 66.134, 42.335, -59.099]
  MoveL 5628 to (-38.66, 42.91, 88.06) mm, rotated rx 180 ry 0 rz 180 deg; joints [-38.016, -26.49, 96.256, 66.134, 42.335, -59.099]
  Call Extruder(65.31188)
  MoveL 5629 to (-38.49, 42.6, 88.06) mm, rotated rx 180 ry 0 rz 180 deg; joints [-37.939, -26.497, 96.26, 66.073, 42.27, -59.052]
  MoveL 5630 to (-38.49, 42.6, 88.06) mm, rotated rx 180 ry 0 rz 180 deg; joints [-37.939, -26.497, 96.26, 66.073, 42.27, -59.052]
  Call Extruder(65.51960)
  MoveL 5631 to (-38.31, 42.3, 88.06) mm, rotated rx 180 ry 0 rz 180 deg; joints [-37.863, -26.503, 96.263, 66.011, 42.206, -59.005]
  MoveL 5632 to (-38.31, 42.3, 88.06) mm, rotated rx 180 ry 0 rz 180 deg; joints [-37.863, -26.503, 96.263, 66.011, 42.206, -59.005]
  Call Extruder(65.72810)
  MoveL 5633 to (-38.14, 41.99, 88.06) mm, rotated rx 180 ry 0 rz -180 deg; joints [-37.787, -26.51, 96.267, 65.95, 42.142, -58.957]
  MoveL 5634 to (-38.14, 41.99, 88.06) mm, rotated rx 180 ry 0 rz -180 deg; joints [-37.787, -26.51, 96.267, 65.95, 42.142, -58.957]
  Call Extruder(65.90765)
  MoveL 5635 to (-37.96, 41.75, 88.06) mm, rotated rx 180 ry 0 rz -180 deg; joints [-37.72, -26.511, 96.267, 65.898, 42.085, -58.919]
  MoveL 5636 to (-37.96, 41.75, 88.06) mm, rotated rx 180 ry 0 rz -180 deg; joints [-37.72, -26.511, 96.267, 65.898, 42.085, -58.919]
  Call Extruder(66.24109)
  MoveL 5637 to (-37.63, 41.3, 88.06) mm, rotated rx -180 ry 0 rz 180 deg; joints [-37.598, -26.513, 96.268, 65.803, 41.981, -58.847]
  MoveL 5638 to (-37.63, 41.3, 88.06) mm, rotated rx -180 ry 0 rz 180 deg; joints [-37.598, -26.513, 96.268, 65.803, 41.981, -58.847]
  Call Extruder(66.57571)
  MoveL 5639 to (-37.3, 40.85, 88.06) mm, rotated rx 180 ry 0 rz 180 deg; joints [-37.475, -26.515, 96.27, 65.707, 41.877, -58.775]
  Call Extruder(67.40364)
  MoveL 5640 to (-36.39, 39.81, 88.06) mm, rotated rx -180 ry 0 rz 180 deg; joints [-37.173, -26.502, 96.263, 65.477, 41.616, -58.607]
  Call Extruder(68.23155)
  MoveL 5641 to (-35.35, 38.9, 88.06) mm, rotated rx 180 ry 0 rz 180 deg; joints [-36.876, -26.465, 96.243, 65.261, 41.355, -58.456]
  Call Extruder(68.39886)
  MoveL 5642 to (-35.13, 38.73, 88.06) mm, rotated rx 180 ry 0 rz 180 deg; joints [-36.818, -26.454, 96.237, 65.219, 41.303, -58.428]
  MoveL 5643 to (-35.13, 38.73, 88.06) mm, rotated rx 180 ry 0 rz 180 deg; joints [-36.818, -26.454, 96.237, 65.219, 41.303, -58.428]
  Call Extruder(68.73228)
  MoveL 5644 to (-34.68, 38.4, 88.06) mm, rotated rx -180 ry 0 rz 180 deg; joints [-36.701, -26.432, 96.225, 65.137, 41.2, -58.372]
  MoveL 5645 to (-34.68, 38.4, 88.06) mm, rotated rx -180 ry 0 rz 180 deg; joints [-36.701, -26.432, 96.225, 65.137, 41.2, -58.372]
  Call Extruder(69.06452)
  MoveL 5646 to (-34.23, 38.08, 88.06) mm, rotated rx 180 ry 0 rz 180 deg; joints [-36.584, -26.41, 96.214, 65.055, 41.096, -58.316]
  MoveL 5647 to (-34.23, 38.08, 88.06) mm, rotated rx 180 ry 0 rz 180 deg; joints [-36.584, -26.41, 96.214, 65.055, 41.096, -58.316]
  Call Extruder(69.18223)
  MoveL 5648 to (-34.05, 37.98, 88.06) mm, rotated rx 180 ry 0 rz 180 deg; joints [-36.544, -26.4, 96.208, 65.028, 41.06, -58.299]
  MoveL 5649 to (-34.05, 37.98, 88.06) mm, rotated rx 180 ry 0 rz 180 deg; joints [-36.544, -26.4, 96.208, 65.028, 41.06, -58.299]
  Call Extruder(69.38995)
  MoveL 5650 to (-33.75, 37.8, 88.06) mm, rotated rx 180 ry 0 rz 180 deg; joints [-36.474, -26.381, 96.198, 64.98, 40.996, -58.268]
  MoveL 5651 to (-33.75, 37.8, 88.06) mm, rotated rx 180 ry 0 rz 180 deg; joints [-36.474, -26.381, 96.198, 64.98, 40.996, -58.268]
  Call Extruder(69.59689)
  MoveL 5652 to (-33.45, 37.63, 88.06) mm, rotated rx 180 ry 0 rz 180 deg; joints [-36.403, -26.363, 96.188, 64.933, 40.933, -58.238]
  MoveL 5653 to (-33.45, 37.63, 88.06) mm, rotated rx 180 ry 0 rz 180 deg; joints [-36.403, -26.363, 96.188, 64.933, 40.933, -58.238]
  Call Extruder(69.80305)
  MoveL 5654 to (-33.14, 37.45, 88.06) mm, rotated rx 180 ry 0 rz 180 deg; joints [-36.333, -26.344, 96.178, 64.886, 40.87, -58.207]
  MoveL 5655 to (-33.14, 37.45, 88.06) mm, rotated rx 180 ry 0 rz 180 deg; joints [-36.333, -26.344, 96.178, 64.886, 40.87, -58.207]
  Call Extruder(69.98473)
  MoveL 5656 to (-32.86, 37.31, 88.06) mm, rotated rx -180 ry 0 rz 180 deg; joints [-36.272, -26.325, 96.168, 64.846, 40.814, -58.182]
  MoveL 5657 to (-32.86, 37.31, 88.06) mm, rotated rx -180 ry 0 rz 180 deg; joints [-36.272, -26.325, 96.168, 64.846, 40.814, -58.182]
  Call Extruder(70.14273)
  MoveL 5658 to (-32.62, 37.2, 88.06) mm, rotated rx 180 ry 0 rz 180 deg; joints [-36.221, -26.307, 96.158, 64.813, 40.767, -58.162]
  MoveL 5659 to (-32.62, 37.2, 88.06) mm, rotated rx 180 ry 0 rz 180 deg; joints [-36.221, -26.307, 96.158, 64.813, 40.767, -58.162]
  Call Extruder(70.30013)
  MoveL 5660 to (-32.37, 37.09, 88.06) mm, rotated rx 180 ry 0 rz 180 deg; joints [-36.17, -26.289, 96.148, 64.781, 40.72, -58.143]
  MoveL 5661 to (-32.37, 37.09, 88.06) mm, rotated rx 180 ry 0 rz 180 deg; joints [-36.17, -26.289, 96.148, 64.781, 40.72, -58.143]
  Call Extruder(70.48284)
  MoveL 5662 to (-32.08, 36.97, 88.06) mm, rotated rx -180 ry 0 rz 180 deg; joints [-36.112, -26.267, 96.137, 64.744, 40.666, -58.121]
  MoveL 5663 to (-32.08, 36.97, 88.06) mm, rotated rx -180 ry 0 rz 180 deg; joints [-36.112, -26.267, 96.137, 64.744, 40.666, -58.121]
  Call Extruder(70.66479)
  MoveL 5664 to (-31.78, 36.85, 88.06) mm, rotated rx -180 ry 0 rz 180 deg; joints [-36.053, -26.245, 96.125, 64.707, 40.612, -58.099]
  MoveL 5665 to (-31.78, 36.85, 88.06) mm, rotated rx -180 ry 0 rz 180 deg; joints [-36.053, -26.245, 96.125, 64.707, 40.612, -58.099]
  Call Extruder(70.81212)
  MoveL 5666 to (-31.54, 36.76, 88.06) mm, rotated rx 180 ry 0 rz 180 deg; joints [-36.006, -26.226, 96.115, 64.678, 40.569, -58.082]
  MoveL 5667 to (-31.54, 36.76, 88.06) mm, rotated rx 180 ry 0 rz 180 deg; joints [-36.006, -26.226, 96.115, 64.678, 40.569, -58.082]
  Call Extruder(70.92536)
  MoveL 5668 to (-31.35, 36.7, 88.06) mm, rotated rx 180 ry 0 rz 180 deg; joints [-35.971, -26.211, 96.106, 64.657, 40.536, -58.07]
  MoveL 5669 to (-31.35, 36.7, 88.06) mm, rotated rx 180 ry 0 rz 180 deg; joints [-35.971, -26.211, 96.106, 64.657, 40.536, -58.07]
  Call Extruder(71.03815)
  MoveL 5670 to (-31.17, 36.64, 88.06) mm, rotated rx 180 ry 0 rz 180 deg; joints [-35.936, -26.195, 96.098, 64.637, 40.503, -58.059]
  MoveL 5671 to (-31.17, 36.64, 88.06) mm, rotated rx 180 ry 0 rz 180 deg; joints [-35.936, -26.195, 96.098, 64.637, 40.503, -58.059]
  Call Extruder(71.15050)
  MoveL 5672 to (-30.98, 36.58, 88.06) mm, rotated rx 180 ry 0 rz -180 deg; joints [-35.901, -26.18, 96.09, 64.616, 40.47, -58.047]
  MoveL 5673 to (-30.98, 36.58, 88.06) mm, rotated rx 180 ry 0 rz -180 deg; joints [-35.901, -26.18, 96.09, 64.616, 40.47, -58.047]
  Call Extruder(71.26240)
  MoveL 5674 to (-30.79, 36.52, 88.06) mm, rotated rx -180 ry 0 rz 180 deg; joints [-35.867, -26.164, 96.081, 64.595, 40.438, -58.035]
  MoveL 5675 to (-30.79, 36.52, 88.06) mm, rotated rx -180 ry 0 rz 180 deg; joints [-35.867, -26.164, 96.081, 64.595, 40.438, -58.035]
  Call Extruder(71.38380)
  MoveL 5676 to (-30.58, 36.45, 88.06) mm, rotated rx 180 ry 0 rz 180 deg; joints [-35.829, -26.147, 96.072, 64.573, 40.403, -58.023]
  MoveL 5677 to (-30.58, 36.45, 88.06) mm, rotated rx 180 ry 0 rz 180 deg; joints [-35.829, -26.147, 96.072, 64.573, 40.403, -58.023]
  Call Extruder(71.51459)
  MoveL 5678 to (-30.36, 36.38, 88.06) mm, rotated rx 180 ry 0 rz 180 deg; joints [-35.788, -26.128, 96.062, 64.549, 40.365, -58.01]
  MoveL 5679 to (-30.36, 36.38, 88.06) mm, rotated rx 180 ry 0 rz 180 deg; joints [-35.788, -26.128, 96.062, 64.549, 40.365, -58.01]
  Call Extruder(71.64482)
  MoveL 5680 to (-30.14, 36.32, 88.06) mm, rotated rx 180 ry 0 rz 180 deg; joints [-35.748, -26.109, 96.052, 64.525, 40.327, -57.997]
  MoveL 5681 to (-30.14, 36.32, 88.06) mm, rotated rx 180 ry 0 rz 180 deg; joints [-35.748, -26.109, 96.052, 64.525, 40.327, -57.997]
  Call Extruder(71.77448)
  MoveL 5682 to (-29.91, 36.25, 88.06) mm, rotated rx 180 ry 0 rz 180 deg; joints [-35.708, -26.09, 96.041, 64.501, 40.289, -57.984]
  MoveL 5683 to (-29.91, 36.25, 88.06) mm, rotated rx 180 ry 0 rz 180 deg; joints [-35.708, -26.09, 96.041, 64.501, 40.289, -57.984]
  Call Extruder(71.90358)
  MoveL 5684 to (-29.69, 36.18, 88.06) mm, rotated rx 180 ry 0 rz 180 deg; joints [-35.668, -26.071, 96.031, 64.478, 40.251, -57.971]
  MoveL 5685 to (-29.69, 36.18, 88.06) mm, rotated rx 180 ry 0 rz 180 deg; joints [-35.668, -26.071, 96.031, 64.478, 40.251, -57.971]
  Call Extruder(72.01865)
  MoveL 5686 to (-29.48, 36.14, 88.06) mm, rotated rx -180 ry 0 rz 180 deg; joints [-35.634, -26.053, 96.021, 64.459, 40.219, -57.962]
  MoveL 5687 to (-29.48, 36.14, 88.06) mm, rotated rx -180 ry 0 rz 180 deg; joints [-35.634, -26.053, 96.021, 64.459, 40.219, -57.962]
  Call Extruder(72.13327)
  MoveL 5688 to (-29.28, 36.09, 88.06) mm, rotated rx 180 ry 0 rz 180 deg; joints [-35.601, -26.034, 96.011, 64.441, 40.187, -57.952]
  MoveL 5689 to (-29.28, 36.09, 88.06) mm, rotated rx 180 ry 0 rz 180 deg; joints [-35.601, -26.034, 96.011, 64.441, 40.187, -57.952]
  Call Extruder(72.24744)
  MoveL 5690 to (-29.08, 36.05, 88.06) mm, rotated rx -180 ry 0 rz 180 deg; joints [-35.567, -26.015, 96.001, 64.422, 40.154, -57.943]
  MoveL 5691 to (-29.08, 36.05, 88.06) mm, rotated rx -180 ry 0 rz 180 deg; joints [-35.567, -26.015, 96.001, 64.422, 40.154, -57.943]
  Call Extruder(72.36115)
  MoveL 5692 to (-28.87, 36, 88.06) mm, rotated rx 180 ry 0 rz 180 deg; joints [-35.533, -25.997, 95.991, 64.404, 40.122, -57.934]
  MoveL 5693 to (-28.87, 36, 88.06) mm, rotated rx 180 ry 0 rz 180 deg; joints [-35.533, -25.997, 95.991, 64.404, 40.122, -57.934]
  Call Extruder(72.48657)
  MoveL 5694 to (-28.64, 35.96, 88.06) mm, rotated rx 180 ry 0 rz 180 deg; joints [-35.497, -25.976, 95.979, 64.384, 40.087, -57.924]
  MoveL 5695 to (-28.64, 35.96, 88.06) mm, rotated rx 180 ry 0 rz 180 deg; joints [-35.497, -25.976, 95.979, 64.384, 40.087, -57.924]
  Call Extruder(72.62355)
  MoveL 5696 to (-28.4, 35.91, 88.06) mm, rotated rx -180 ry 0 rz 180 deg; joints [-35.457, -25.953, 95.967, 64.362, 40.048, -57.914]
  MoveL 5697 to (-28.4, 35.91, 88.06) mm, rotated rx -180 ry 0 rz 180 deg; joints [-35.457, -25.953, 95.967, 64.362, 40.048, -57.914]
  Call Extruder(72.75992)
  MoveL 5698 to (-28.15, 35.86, 88.06) mm, rotated rx 180 ry 0 rz 180 deg; joints [-35.417, -25.929, 95.954, 64.34, 40.01, -57.904]
  MoveL 5699 to (-28.15, 35.86, 88.06) mm, rotated rx 180 ry 0 rz 180 deg; joints [-35.417, -25.929, 95.954, 64.34, 40.01, -57.904]
  Call Extruder(72.89567)
  MoveL 5700 to (-27.9, 35.81, 88.06) mm, rotated rx 180 ry 0 rz 180 deg; joints [-35.377, -25.906, 95.942, 64.319, 39.972, -57.893]
  MoveL 5701 to (-27.9, 35.81, 88.06) mm, rotated rx 180 ry 0 rz 180 deg; joints [-35.377, -25.906, 95.942, 64.319, 39.972, -57.893]
  Call Extruder(73.03082)
  MoveL 5702 to (-27.65, 35.76, 88.06) mm, rotated rx -180 ry 0 rz 180 deg; joints [-35.337, -25.883, 95.929, 64.297, 39.933, -57.883]
  MoveL 5703 to (-27.65, 35.76, 88.06) mm, rotated rx -180 ry 0 rz 180 deg; joints [-35.337, -25.883, 95.929, 64.297, 39.933, -57.883]
  Call Extruder(73.16536)
  MoveL 5704 to (-27.4, 35.71, 88.06) mm, rotated rx -180 ry 0 rz 180 deg; joints [-35.297, -25.86, 95.916, 64.276, 39.895, -57.872]
  MoveL 5705 to (-27.4, 35.71, 88.06) mm, rotated rx -180 ry 0 rz 180 deg; joints [-35.297, -25.86, 95.916, 64.276, 39.895, -57.872]
  Call Extruder(73.29928)
  MoveL 5706 to (-27.15, 35.66, 88.06) mm, rotated rx 180 ry 0 rz 180 deg; joints [-35.258, -25.836, 95.903, 64.254, 39.857, -57.862]
  MoveL 5707 to (-27.15, 35.66, 88.06) mm, rotated rx 180 ry 0 rz 180 deg; joints [-35.258, -25.836, 95.903, 64.254, 39.857, -57.862]
  Call Extruder(73.44714)
  MoveL 5708 to (-26.87, 35.61, 88.06) mm, rotated rx 180 ry 0 rz 180 deg; joints [-35.215, -25.81, 95.889, 64.231, 39.815, -57.851]
  MoveL 5709 to (-26.87, 35.61, 88.06) mm, rotated rx 180 ry 0 rz 180 deg; joints [-35.215, -25.81, 95.889, 64.231, 39.815, -57.851]
  Call Extruder(73.60888)
  MoveL 5710 to (-26.57, 35.56, 88.06) mm, rotated rx 180 ry 0 rz -180 deg; joints [-35.168, -25.78, 95.873, 64.207, 39.77, -57.841]
  MoveL 5711 to (-26.57, 35.56, 88.06) mm, rotated rx 180 ry 0 rz -180 deg; joints [-35.168, -25.78, 95.873, 64.207, 39.77, -57.841]
  Call Extruder(73.76989)
  MoveL 5712 to (-26.26, 35.51, 88.06) mm, rotated rx -180 ry 0 rz -180 deg; joints [-35.122, -25.751, 95.857, 64.183, 39.725, -57.83]
  MoveL 5713 to (-26.26, 35.51, 88.06) mm, rotated rx -180 ry 0 rz -180 deg; joints [-35.122, -25.751, 95.857, 64.183, 39.725, -57.83]
  Call Extruder(73.93017)
  MoveL 5714 to (-25.96, 35.47, 88.06) mm, rotated rx 180 ry 0 rz 180 deg; joints [-35.075, -25.721, 95.84, 64.159, 39.68, -57.819]
  MoveL 5715 to (-25.96, 35.47, 88.06) mm, rotated rx 180 ry 0 rz 180 deg; joints [-35.075, -25.721, 95.84, 64.159, 39.68, -57.819]
  Call Extruder(74.08972)
  MoveL 5716 to (-25.65, 35.42, 88.06) mm, rotated rx 180 ry 0 rz 180 deg; joints [-35.029, -25.691, 95.824, 64.135, 39.635, -57.808]
  MoveL 5717 to (-25.65, 35.42, 88.06) mm, rotated rx 180 ry 0 rz 180 deg; joints [-35.029, -25.691, 95.824, 64.135, 39.635, -57.808]
  Call Extruder(74.24855)
  MoveL 5718 to (-25.34, 35.37, 88.06) mm, rotated rx -180 ry 0 rz 180 deg; joints [-34.983, -25.662, 95.808, 64.111, 39.59, -57.797]
  MoveL 5719 to (-25.34, 35.37, 88.06) mm, rotated rx -180 ry 0 rz 180 deg; joints [-34.983, -25.662, 95.808, 64.111, 39.59, -57.797]
  Call Extruder(74.42721)
  MoveL 5720 to (-25, 35.32, 88.06) mm, rotated rx 180 ry 0 rz 180 deg; joints [-34.932, -25.627, 95.789, 64.085, 39.54, -57.787]
  MoveL 5721 to (-25, 35.32, 88.06) mm, rotated rx 180 ry 0 rz 180 deg; joints [-34.932, -25.627, 95.789, 64.085, 39.54, -57.787]
  Call Extruder(74.62566)
  MoveL 5722 to (-24.61, 35.28, 88.06) mm, rotated rx 180 ry 0 rz 180 deg; joints [-34.877, -25.588, 95.768, 64.058, 39.486, -57.775]
  MoveL 5723 to (-24.61, 35.28, 88.06) mm, rotated rx 180 ry 0 rz 180 deg; joints [-34.877, -25.588, 95.768, 64.058, 39.486, -57.775]
  Call Extruder(74.82323)
  MoveL 5724 to (-24.22, 35.23, 88.06) mm, rotated rx -180 ry 0 rz 180 deg; joints [-34.821, -25.55, 95.746, 64.031, 39.431, -57.764]
  MoveL 5725 to (-24.22, 35.23, 88.06) mm, rotated rx -180 ry 0 rz 180 deg; joints [-34.821, -25.55, 95.746, 64.031, 39.431, -57.764]
  Call Extruder(75.01994)
  MoveL 5726 to (-23.84, 35.18, 88.06) mm, rotated rx -180 ry 0 rz -180 deg; joints [-34.766, -25.51, 95.725, 64.003, 39.377, -57.753]
  MoveL 5727 to (-23.84, 35.18, 88.06) mm, rotated rx -180 ry 0 rz -180 deg; joints [-34.766, -25.51, 95.725, 64.003, 39.377, -57.753]
  Call Extruder(75.21578)
  MoveL 5728 to (-23.45, 35.14, 88.06) mm, rotated rx -180 ry 0 rz 180 deg; joints [-34.711, -25.471, 95.703, 63.976, 39.323, -57.742]
  MoveL 5729 to (-23.45, 35.14, 88.06) mm, rotated rx -180 ry 0 rz 180 deg; joints [-34.711, -25.471, 95.703, 63.976, 39.323, -57.742]
  Call Extruder(75.51117)
  MoveL 5730 to (-22.86, 35.09, 88.06) mm, rotated rx 180 ry 0 rz 180 deg; joints [-34.631, -25.41, 95.669, 63.939, 39.243, -57.729]
  MoveL 5731 to (-22.86, 35.09, 88.06) mm, rotated rx 180 ry 0 rz 180 deg; joints [-34.631, -25.41, 95.669, 63.939, 39.243, -57.729]
  Call Extruder(75.80523)
  MoveL 5732 to (-22.27, 35.05, 88.06) mm, rotated rx 180 ry 0 rz 180 deg; joints [-34.552, -25.349, 95.635, 63.902, 39.164, -57.716]
  MoveL 5733 to (-22.27, 35.05, 88.06) mm, rotated rx 180 ry 0 rz 180 deg; joints [-34.552, -25.349, 95.635, 63.902, 39.164, -57.716]
  Call Extruder(76.09796)
  MoveL 5734 to (-21.68, 35, 88.06) mm, rotated rx -180 ry 0 rz 180 deg; joints [-34.473, -25.287, 95.601, 63.865, 39.085, -57.703]
  MoveL 5735 to (-21.68, 35, 88.06) mm, rotated rx -180 ry 0 rz 180 deg; joints [-34.473, -25.287, 95.601, 63.865, 39.085, -57.703]
  Call Extruder(76.67141)
  MoveL 5736 to (-20.52, 34.95, 88.06) mm, rotated rx 180 ry 0 rz 180 deg; joints [-34.326, -25.162, 95.532, 63.802, 38.937, -57.685]
  MoveL 5737 to (-20.52, 34.95, 88.06) mm, rotated rx 180 ry 0 rz 180 deg; joints [-34.326, -25.162, 95.532, 63.802, 38.937, -57.685]
  Call Extruder(77.38537)
  MoveL 5738 to (-19.06, 34.91, 88.06) mm, rotated rx 180 ry 0 rz 180 deg; joints [-34.146, -25.004, 95.443, 63.726, 38.754, -57.665]
  Call Extruder(194.23211)
  MoveL 5739 to (219.06, 34.91, 88.06) mm, rotated rx -180 ry 0 rz -180 deg; joints [-18.248, 6.847, 68.612, 52.712, 23.178, -50.365]
  Call Extruder(194.66067)
  MoveL 5740 to (219.94, 34.93, 88.06) mm, rotated rx -180 ry 0 rz 180 deg; joints [-18.218, 6.988, 68.455, 52.632, 23.165, -50.286]
  MoveL 5741 to (219.94, 34.93, 88.06) mm, rotated rx -180 ry 0 rz 180 deg; joints [-18.218, 6.988, 68.455, 52.632, 23.165, -50.286]
  Call Extruder(195.23412)
  MoveL 5742 to (221.1, 34.97, 88.06) mm, rotated rx 180 ry 0 rz 180 deg; joints [-18.181, 7.177, 68.243, 52.529, 23.15, -50.183]
  MoveL 5743 to (221.1, 34.97, 88.06) mm, rotated rx 180 ry 0 rz 180 deg; joints [-18.181, 7.177, 68.243, 52.529, 23.15, -50.183]
  Call Extruder(195.66843)
  MoveL 5744 to (221.97, 35.02, 88.06) mm, rotated rx 180 ry 0 rz -180 deg; joints [-18.154, 7.32, 68.081, 52.452, 23.14, -50.107]
  MoveL 5745 to (221.97, 35.02, 88.06) mm, rotated rx 180 ry 0 rz -180 deg; joints [-18.154, 7.32, 68.081, 52.452, 23.14, -50.107]
  Call Extruder(195.96249)
  MoveL 5746 to (222.56, 35.07, 88.06) mm, rotated rx 180 ry 0 rz -180 deg; joints [-18.138, 7.418, 67.972, 52.402, 23.135, -50.058]
  MoveL 5747 to (222.56, 35.07, 88.06) mm, rotated rx 180 ry 0 rz -180 deg; joints [-18.138, 7.418, 67.972, 52.402, 23.135, -50.058]
  Call Extruder(196.25788)
  MoveL 5748 to (223.15, 35.11, 88.06) mm, rotated rx 180 ry 0 rz -180 deg; joints [-18.121, 7.515, 67.862, 52.352, 23.13, -50.008]
  MoveL 5749 to (223.15, 35.11, 88.06) mm, rotated rx 180 ry 0 rz -180 deg; joints [-18.121, 7.515, 67.862, 52.352, 23.13, -50.008]
  Call Extruder(196.50411)
  MoveL 5750 to (223.64, 35.16, 88.06) mm, rotated rx -180 ry 0 rz 180 deg; joints [-18.109, 7.596, 67.77, 52.312, 23.127, -49.968]
  MoveL 5751 to (223.64, 35.16, 88.06) mm, rotated rx -180 ry 0 rz 180 deg; joints [-18.109, 7.596, 67.77, 52.312, 23.127, -49.968]
  Call Extruder(196.70082)
  MoveL 5752 to (224.03, 35.21, 88.06) mm, rotated rx -180 ry 0 rz -180 deg; joints [-18.1, 7.662, 67.696, 52.282, 23.126, -49.937]
  MoveL 5753 to (224.03, 35.21, 88.06) mm, rotated rx -180 ry 0 rz -180 deg; joints [-18.1, 7.662, 67.696, 52.282, 23.126, -49.937]
  Call Extruder(196.89840)
  MoveL 5754 to (224.42, 35.25, 88.06) mm, rotated rx 180 ry 0 rz 180 deg; joints [-18.091, 7.727, 67.622, 52.251, 23.124, -49.906]
  MoveL 5755 to (224.42, 35.25, 88.06) mm, rotated rx 180 ry 0 rz 180 deg; joints [-18.091, 7.727, 67.622, 52.251, 23.124, -49.906]
  Call Extruder(197.09684)
  MoveL 5756 to (224.8, 35.3, 88.06) mm, rotated rx 180 ry 0 rz 180 deg; joints [-18.082, 7.792, 67.548, 52.221, 23.123, -49.875]
  MoveL 5757 to (224.8, 35.3, 88.06) mm, rotated rx 180 ry 0 rz 180 deg; joints [-18.082, 7.792, 67.548, 52.221, 23.123, -49.875]
  Call Extruder(197.29615)
  MoveL 5758 to (225.19, 35.34, 88.06) mm, rotated rx -180 ry 0 rz 180 deg; joints [-18.073, 7.857, 67.475, 52.19, 23.121, -49.844]
  MoveL 5759 to (225.19, 35.34, 88.06) mm, rotated rx -180 ry 0 rz 180 deg; joints [-18.073, 7.857, 67.475, 52.19, 23.121, -49.844]
  Call Extruder(197.45497)
  MoveL 5760 to (225.5, 35.39, 88.06) mm, rotated rx -180 ry 0 rz 180 deg; joints [-18.068, 7.909, 67.415, 52.167, 23.121, -49.822]
  MoveL 5761 to (225.5, 35.39, 88.06) mm, rotated rx -180 ry 0 rz 180 deg; joints [-18.068, 7.909, 67.415, 52.167, 23.121, -49.822]
  Call Extruder(197.61452)
  MoveL 5762 to (225.8, 35.44, 88.06) mm, rotated rx 180 ry 0 rz -180 deg; joints [-18.062, 7.961, 67.356, 52.145, 23.121, -49.799]
  MoveL 5763 to (225.8, 35.44, 88.06) mm, rotated rx 180 ry 0 rz -180 deg; joints [-18.062, 7.961, 67.356, 52.145, 23.121, -49.799]
  Call Extruder(197.77480)
  MoveL 5764 to (226.11, 35.49, 88.06) mm, rotated rx 180 ry 0 rz 180 deg; joints [-18.056, 8.014, 67.297, 52.122, 23.121, -49.776]
  MoveL 5765 to (226.11, 35.49, 88.06) mm, rotated rx 180 ry 0 rz 180 deg; joints [-18.056, 8.014, 67.297, 52.122, 23.121, -49.776]
  Call Extruder(197.93580)
  MoveL 5766 to (226.41, 35.54, 88.06) mm, rotated rx 180 ry 0 rz 180 deg; joints [-18.051, 8.066, 67.237, 52.1, 23.122, -49.753]
  MoveL 5767 to (226.41, 35.54, 88.06) mm, rotated rx 180 ry 0 rz 180 deg; joints [-18.051, 8.066, 67.237, 52.1, 23.122, -49.753]
  Call Extruder(198.09753)
  MoveL 5768 to (226.72, 35.59, 88.06) mm, rotated rx -180 ry 0 rz -180 deg; joints [-18.045, 8.118, 67.177, 52.077, 23.122, -49.729]
  MoveL 5769 to (226.72, 35.59, 88.06) mm, rotated rx -180 ry 0 rz -180 deg; joints [-18.045, 8.118, 67.177, 52.077, 23.122, -49.729]
  Call Extruder(198.25999)
  MoveL 5770 to (227.02, 35.64, 88.06) mm, rotated rx 180 ry 0 rz 180 deg; joints [-18.039, 8.17, 67.118, 52.054, 23.122, -49.706]
  MoveL 5771 to (227.02, 35.64, 88.06) mm, rotated rx 180 ry 0 rz 180 deg; joints [-18.039, 8.17, 67.118, 52.054, 23.122, -49.706]
  Call Extruder(198.39392)
  MoveL 5772 to (227.27, 35.68, 88.06) mm, rotated rx 180 ry 0 rz -180 deg; joints [-18.036, 8.214, 67.069, 52.037, 23.123, -49.689]
  MoveL 5773 to (227.27, 35.68, 88.06) mm, rotated rx 180 ry 0 rz -180 deg; joints [-18.036, 8.214, 67.069, 52.037, 23.123, -49.689]
  Call Extruder(198.52846)
  MoveL 5774 to (227.52, 35.73, 88.06) mm, rotated rx 180 ry 0 rz -180 deg; joints [-18.033, 8.257, 67.019, 52.02, 23.124, -49.671]
  MoveL 5775 to (227.52, 35.73, 88.06) mm, rotated rx 180 ry 0 rz -180 deg; joints [-18.033, 8.257, 67.019, 52.02, 23.124, -49.671]
  Call Extruder(198.66360)
  MoveL 5776 to (227.77, 35.78, 88.06) mm, rotated rx -180 ry 0 rz -180 deg; joints [-18.029, 8.3, 66.97, 52.003, 23.125, -49.654]
  MoveL 5777 to (227.77, 35.78, 88.06) mm, rotated rx -180 ry 0 rz -180 deg; joints [-18.029, 8.3, 66.97, 52.003, 23.125, -49.654]
  Call Extruder(198.79936)
  MoveL 5778 to (228.02, 35.83, 88.06) mm, rotated rx 180 ry 0 rz -180 deg; joints [-18.026, 8.343, 66.92, 51.986, 23.126, -49.636]
  MoveL 5779 to (228.02, 35.83, 88.06) mm, rotated rx 180 ry 0 rz -180 deg; joints [-18.026, 8.343, 66.92, 51.986, 23.126, -49.636]
  Call Extruder(198.93573)
  MoveL 5780 to (228.27, 35.88, 88.06) mm, rotated rx 180 ry 0 rz 180 deg; joints [-18.022, 8.387, 66.871, 51.969, 23.128, -49.618]
  MoveL 5781 to (228.27, 35.88, 88.06) mm, rotated rx 180 ry 0 rz 180 deg; joints [-18.022, 8.387, 66.871, 51.969, 23.128, -49.618]
  Call Extruder(199.07271)
  MoveL 5782 to (228.52, 35.93, 88.06) mm, rotated rx -180 ry 0 rz 180 deg; joints [-18.019, 8.43, 66.821, 51.952, 23.129, -49.6]
  MoveL 5783 to (228.52, 35.93, 88.06) mm, rotated rx -180 ry 0 rz 180 deg; joints [-18.019, 8.43, 66.821, 51.952, 23.129, -49.6]
  Call Extruder(199.21030)
  MoveL 5784 to (228.77, 35.98, 88.06) mm, rotated rx 180 ry 0 rz 180 deg; joints [-18.015, 8.473, 66.772, 51.934, 23.13, -49.583]
  MoveL 5785 to (228.77, 35.98, 88.06) mm, rotated rx 180 ry 0 rz 180 deg; joints [-18.015, 8.473, 66.772, 51.934, 23.13, -49.583]
  Call Extruder(199.32402)
  MoveL 5786 to (228.97, 36.03, 88.06) mm, rotated rx -180 ry 0 rz -180 deg; joints [-18.013, 8.509, 66.731, 51.921, 23.132, -49.568]
  MoveL 5787 to (228.97, 36.03, 88.06) mm, rotated rx -180 ry 0 rz -180 deg; joints [-18.013, 8.509, 66.731, 51.921, 23.132, -49.568]
  Call Extruder(199.43819)
  MoveL 5788 to (229.18, 36.07, 88.06) mm, rotated rx -180 ry 0 rz 180 deg; joints [-18.01, 8.545, 66.689, 51.907, 23.133, -49.554]
  MoveL 5789 to (229.18, 36.07, 88.06) mm, rotated rx -180 ry 0 rz 180 deg; joints [-18.01, 8.545, 66.689, 51.907, 23.133, -49.554]
  Call Extruder(199.55281)
  MoveL 5790 to (229.38, 36.12, 88.06) mm, rotated rx -180 ry 0 rz 180 deg; joints [-18.008, 8.581, 66.648, 51.893, 23.135, -49.54]
  MoveL 5791 to (229.38, 36.12, 88.06) mm, rotated rx -180 ry 0 rz 180 deg; joints [-18.008, 8.581, 66.648, 51.893, 23.135, -49.54]
  Call Extruder(199.66788)
  MoveL 5792 to (229.59, 36.16, 88.06) mm, rotated rx -180 ry 0 rz 180 deg; joints [-18.006, 8.617, 66.607, 51.88, 23.136, -49.526]
  MoveL 5793 to (229.59, 36.16, 88.06) mm, rotated rx -180 ry 0 rz 180 deg; joints [-18.006, 8.617, 66.607, 51.88, 23.136, -49.526]
  Call Extruder(199.79012)
  MoveL 5794 to (229.8, 36.22, 88.06) mm, rotated rx 180 ry 0 rz 180 deg; joints [-18.004, 8.655, 66.564, 51.867, 23.138, -49.512]
  MoveL 5795 to (229.8, 36.22, 88.06) mm, rotated rx 180 ry 0 rz 180 deg; joints [-18.004, 8.655, 66.564, 51.867, 23.138, -49.512]
  Call Extruder(199.91978)
  MoveL 5796 to (230.02, 36.28, 88.06) mm, rotated rx 180 ry 0 rz 180 deg; joints [-18.004, 8.695, 66.517, 51.855, 23.142, -49.499]
  MoveL 5797 to (230.02, 36.28, 88.06) mm, rotated rx 180 ry 0 rz 180 deg; joints [-18.004, 8.695, 66.517, 51.855, 23.142, -49.499]
  Call Extruder(200.05001)
  MoveL 5798 to (230.25, 36.35, 88.06) mm, rotated rx -180 ry 0 rz 180 deg; joints [-18.003, 8.735, 66.471, 51.843, 23.145, -49.487]
  MoveL 5799 to (230.25, 36.35, 88.06) mm, rotated rx -180 ry 0 rz 180 deg; joints [-18.003, 8.735, 66.471, 51.843, 23.145, -49.487]
  Call Extruder(200.18081)
  MoveL 5800 to (230.47, 36.42, 88.06) mm, rotated rx -180 ry 0 rz 180 deg; joints [-18.003, 8.776, 66.425, 51.831, 23.148, -49.474]
  MoveL 5801 to (230.47, 36.42, 88.06) mm, rotated rx -180 ry 0 rz 180 deg; joints [-18.003, 8.776, 66.425, 51.831, 23.148, -49.474]
  Call Extruder(200.31217)
  MoveL 5802 to (230.69, 36.49, 88.06) mm, rotated rx 180 ry 0 rz 180 deg; joints [-18.002, 8.816, 66.378, 51.819, 23.152, -49.461]
  MoveL 5803 to (230.69, 36.49, 88.06) mm, rotated rx 180 ry 0 rz 180 deg; joints [-18.002, 8.816, 66.378, 51.819, 23.152, -49.461]
  Call Extruder(200.40859)
  MoveL 5804 to (230.86, 36.54, 88.06) mm, rotated rx -180 ry 0 rz -180 deg; joints [-18.002, 8.845, 66.344, 51.81, 23.154, -49.452]
  MoveL 5805 to (230.86, 36.54, 88.06) mm, rotated rx -180 ry 0 rz -180 deg; joints [-18.002, 8.845, 66.344, 51.81, 23.154, -49.452]
  Call Extruder(200.52476)
  MoveL 5806 to (231.05, 36.6, 88.06) mm, rotated rx 180 ry 0 rz 180 deg; joints [-18.002, 8.881, 66.303, 51.8, 23.158, -49.441]
  MoveL 5807 to (231.05, 36.6, 88.06) mm, rotated rx 180 ry 0 rz 180 deg; joints [-18.002, 8.881, 66.303, 51.8, 23.158, -49.441]
  Call Extruder(200.64140)
  MoveL 5808 to (231.25, 36.67, 88.06) mm, rotated rx -180 ry 0 rz 180 deg; joints [-18.002, 8.916, 66.263, 51.79, 23.161, -49.43]
  MoveL 5809 to (231.25, 36.67, 88.06) mm, rotated rx -180 ry 0 rz 180 deg; joints [-18.002, 8.916, 66.263, 51.79, 23.161, -49.43]
  Call Extruder(200.75852)
  MoveL 5810 to (231.44, 36.73, 88.06) mm, rotated rx 180 ry 0 rz 180 deg; joints [-18.002, 8.952, 66.222, 51.781, 23.164, -49.419]
  MoveL 5811 to (231.44, 36.73, 88.06) mm, rotated rx 180 ry 0 rz 180 deg; joints [-18.002, 8.952, 66.222, 51.781, 23.164, -49.419]
  Call Extruder(200.87612)
  MoveL 5812 to (231.64, 36.79, 88.06) mm, rotated rx 180 ry 0 rz 180 deg; joints [-18.002, 8.987, 66.181, 51.77, 23.168, -49.408]
  MoveL 5813 to (231.64, 36.79, 88.06) mm, rotated rx 180 ry 0 rz 180 deg; joints [-18.002, 8.987, 66.181, 51.77, 23.168, -49.408]
  Call Extruder(201.05807)
  MoveL 5814 to (231.93, 36.91, 88.06) mm, rotated rx -180 ry 0 rz -180 deg; joints [-18.005, 9.042, 66.118, 51.76, 23.175, -49.395]
  MoveL 5815 to (231.93, 36.91, 88.06) mm, rotated rx -180 ry 0 rz -180 deg; joints [-18.005, 9.042, 66.118, 51.76, 23.175, -49.395]
  Call Extruder(201.24079)
  MoveL 5816 to (232.22, 37.04, 88.06) mm, rotated rx 180 ry 0 rz 180 deg; joints [-18.008, 9.096, 66.054, 51.749, 23.183, -49.383]
  MoveL 5817 to (232.22, 37.04, 88.06) mm, rotated rx 180 ry 0 rz 180 deg; joints [-18.008, 9.096, 66.054, 51.749, 23.183, -49.383]
  Call Extruder(201.41121)
  MoveL 5818 to (232.49, 37.15, 88.06) mm, rotated rx -180 ry 0 rz 180 deg; joints [-18.011, 9.147, 65.996, 51.739, 23.19, -49.371]
  MoveL 5819 to (232.49, 37.15, 88.06) mm, rotated rx -180 ry 0 rz 180 deg; joints [-18.011, 9.147, 65.996, 51.739, 23.19, -49.371]
  Call Extruder(201.56921)
  MoveL 5820 to (232.74, 37.26, 88.06) mm, rotated rx -180 ry 0 rz 180 deg; joints [-18.013, 9.194, 65.942, 51.73, 23.197, -49.361]
  MoveL 5821 to (232.74, 37.26, 88.06) mm, rotated rx -180 ry 0 rz 180 deg; joints [-18.013, 9.194, 65.942, 51.73, 23.197, -49.361]
  Call Extruder(201.72781)
  MoveL 5822 to (232.99, 37.36, 88.06) mm, rotated rx -180 ry 0 rz 180 deg; joints [-18.016, 9.241, 65.887, 51.721, 23.203, -49.35]
  MoveL 5823 to (232.99, 37.36, 88.06) mm, rotated rx -180 ry 0 rz 180 deg; joints [-18.016, 9.241, 65.887, 51.721, 23.203, -49.35]
  Call Extruder(201.93398)
  MoveL 5824 to (233.29, 37.54, 88.06) mm, rotated rx -180 ry 0 rz 180 deg; joints [-18.024, 9.3, 65.818, 51.717, 23.215, -49.344]
  MoveL 5825 to (233.29, 37.54, 88.06) mm, rotated rx -180 ry 0 rz 180 deg; joints [-18.024, 9.3, 65.818, 51.717, 23.215, -49.344]
  Call Extruder(202.14092)
  MoveL 5826 to (233.6, 37.71, 88.06) mm, rotated rx -180 ry 0 rz 180 deg; joints [-18.033, 9.36, 65.749, 51.713, 23.228, -49.337]
  MoveL 5827 to (233.6, 37.71, 88.06) mm, rotated rx -180 ry 0 rz 180 deg; joints [-18.033, 9.36, 65.749, 51.713, 23.228, -49.337]
  Call Extruder(202.34865)
  MoveL 5828 to (233.9, 37.89, 88.06) mm, rotated rx 180 ry 0 rz 180 deg; joints [-18.041, 9.42, 65.679, 51.709, 23.24, -49.331]
  MoveL 5829 to (233.9, 37.89, 88.06) mm, rotated rx 180 ry 0 rz 180 deg; joints [-18.041, 9.42, 65.679, 51.709, 23.24, -49.331]
  Call Extruder(202.55715)
  MoveL 5830 to (234.21, 38.07, 88.06) mm, rotated rx -180 ry 0 rz -180 deg; joints [-18.049, 9.48, 65.61, 51.705, 23.252, -49.324]
  MoveL 5831 to (234.21, 38.07, 88.06) mm, rotated rx -180 ry 0 rz -180 deg; joints [-18.049, 9.48, 65.61, 51.705, 23.252, -49.324]
  Call Extruder(202.73669)
  MoveL 5832 to (234.45, 38.24, 88.06) mm, rotated rx -180 ry 0 rz -180 deg; joints [-18.06, 9.53, 65.551, 51.707, 23.265, -49.323]
  MoveL 5833 to (234.45, 38.24, 88.06) mm, rotated rx -180 ry 0 rz -180 deg; joints [-18.06, 9.53, 65.551, 51.707, 23.265, -49.323]
  Call Extruder(203.07011)
  MoveL 5834 to (234.9, 38.57, 88.06) mm, rotated rx -180 ry 0 rz 180 deg; joints [-18.079, 9.622, 65.444, 51.712, 23.29, -49.323]
  MoveL 5835 to (234.9, 38.57, 88.06) mm, rotated rx -180 ry 0 rz 180 deg; joints [-18.079, 9.622, 65.444, 51.712, 23.29, -49.323]
  Call Extruder(203.40471)
  MoveL 5836 to (235.35, 38.9, 88.06) mm, rotated rx -180 ry 0 rz 180 deg; joints [-18.099, 9.715, 65.335, 51.716, 23.314, -49.321]
  Call Extruder(204.23266)
  MoveL 5837 to (236.39, 39.81, 88.06) mm, rotated rx -180 ry 0 rz 180 deg; joints [-18.16, 9.938, 65.075, 51.749, 23.384, -49.34]
  Call Extruder(205.06060)
  MoveL 5838 to (237.3, 40.85, 88.06) mm, rotated rx -180 ry 0 rz 180 deg; joints [-18.24, 10.147, 64.83, 51.813, 23.466, -49.388]
  Call Extruder(205.22791)
  MoveL 5839 to (237.47, 41.07, 88.06) mm, rotated rx 180 ry 0 rz 180 deg; joints [-18.258, 10.186, 64.783, 51.83, 23.485, -49.401]
  MoveL 5840 to (237.47, 41.07, 88.06) mm, rotated rx 180 ry 0 rz 180 deg; joints [-18.258, 10.186, 64.783, 51.83, 23.485, -49.401]
  Call Extruder(205.56133)
  MoveL 5841 to (237.8, 41.52, 88.06) mm, rotated rx -180 ry 0 rz 180 deg; joints [-18.295, 10.266, 64.689, 51.865, 23.521, -49.429]
  MoveL 5842 to (237.8, 41.52, 88.06) mm, rotated rx -180 ry 0 rz 180 deg; joints [-18.295, 10.266, 64.689, 51.865, 23.521, -49.429]
  Call Extruder(205.89358)
  MoveL 5843 to (238.12, 41.98, 88.06) mm, rotated rx 180 ry 0 rz 180 deg; joints [-18.332, 10.346, 64.595, 51.899, 23.558, -49.456]
  MoveL 5844 to (238.12, 41.98, 88.06) mm, rotated rx 180 ry 0 rz 180 deg; joints [-18.332, 10.346, 64.595, 51.899, 23.558, -49.456]
  Call Extruder(206.06099)
  MoveL 5845 to (238.27, 42.22, 88.06) mm, rotated rx -180 ry 0 rz 180 deg; joints [-18.352, 10.384, 64.551, 51.921, 23.578, -49.473]
  MoveL 5846 to (238.27, 42.22, 88.06) mm, rotated rx -180 ry 0 rz 180 deg; joints [-18.352, 10.384, 64.551, 51.921, 23.578, -49.473]
  Call Extruder(206.21452)
  MoveL 5847 to (238.4, 42.44, 88.06) mm, rotated rx 180 ry 0 rz 180 deg; joints [-18.371, 10.419, 64.51, 51.94, 23.596, -49.489]
  MoveL 5848 to (238.4, 42.44, 88.06) mm, rotated rx 180 ry 0 rz 180 deg; joints [-18.371, 10.419, 64.51, 51.94, 23.596, -49.489]
  Call Extruder(206.42306)
  MoveL 5849 to (238.58, 42.75, 88.06) mm, rotated rx 180 ry 0 rz 180 deg; joints [-18.398, 10.465, 64.455, 51.969, 23.622, -49.513]
  MoveL 5850 to (238.58, 42.75, 88.06) mm, rotated rx 180 ry 0 rz 180 deg; joints [-18.398, 10.465, 64.455, 51.969, 23.622, -49.513]
  Call Extruder(206.63087)
  MoveL 5851 to (238.75, 43.06, 88.06) mm, rotated rx 180 ry 0 rz 180 deg; joints [-18.425, 10.511, 64.4, 51.997, 23.647, -49.536]
  MoveL 5852 to (238.75, 43.06, 88.06) mm, rotated rx 180 ry 0 rz 180 deg; joints [-18.425, 10.511, 64.4, 51.997, 23.647, -49.536]
  Call Extruder(206.81346)
  MoveL 5853 to (238.89, 43.34, 88.06) mm, rotated rx 180 ry 0 rz 180 deg; joints [-18.45, 10.551, 64.354, 52.024, 23.671, -49.559]
  MoveL 5854 to (238.89, 43.34, 88.06) mm, rotated rx 180 ry 0 rz 180 deg; joints [-18.45, 10.551, 64.354, 52.024, 23.671, -49.559]
  Call Extruder(206.97148)
  MoveL 5855 to (239, 43.58, 88.06) mm, rotated rx 180 ry 0 rz 180 deg; joints [-18.472, 10.583, 64.316, 52.05, 23.691, -49.581]
  MoveL 5856 to (239, 43.58, 88.06) mm, rotated rx 180 ry 0 rz 180 deg; joints [-18.472, 10.583, 64.316, 52.05, 23.691, -49.581]
  Call Extruder(207.12890)
  MoveL 5857 to (239.1, 43.83, 88.06) mm, rotated rx -180 ry 0 rz -180 deg; joints [-18.495, 10.615, 64.278, 52.077, 23.712, -49.603]
  MoveL 5858 to (239.1, 43.83, 88.06) mm, rotated rx -180 ry 0 rz -180 deg; joints [-18.495, 10.615, 64.278, 52.077, 23.712, -49.603]
  Call Extruder(207.31161)
  MoveL 5859 to (239.23, 44.13, 88.06) mm, rotated rx 180 ry 0 rz 180 deg; joints [-18.522, 10.651, 64.235, 52.108, 23.737, -49.629]
  MoveL 5860 to (239.23, 44.13, 88.06) mm, rotated rx 180 ry 0 rz 180 deg; joints [-18.522, 10.651, 64.235, 52.108, 23.737, -49.629]
  Call Extruder(207.49357)
  MoveL 5861 to (239.35, 44.42, 88.06) mm, rotated rx 180 ry 0 rz 180 deg; joints [-18.549, 10.688, 64.192, 52.139, 23.761, -49.655]
  MoveL 5862 to (239.35, 44.42, 88.06) mm, rotated rx 180 ry 0 rz 180 deg; joints [-18.549, 10.688, 64.192, 52.139, 23.761, -49.655]
  Call Extruder(207.64090)
  MoveL 5863 to (239.44, 44.66, 88.06) mm, rotated rx -180 ry 0 rz -180 deg; joints [-18.571, 10.717, 64.157, 52.165, 23.782, -49.678]
  MoveL 5864 to (239.44, 44.66, 88.06) mm, rotated rx -180 ry 0 rz -180 deg; joints [-18.571, 10.717, 64.157, 52.165, 23.782, -49.678]
  Call Extruder(207.75414)
  MoveL 5865 to (239.5, 44.85, 88.06) mm, rotated rx 180 ry 0 rz 180 deg; joints [-18.589, 10.738, 64.132, 52.187, 23.798, -49.696]
  MoveL 5866 to (239.5, 44.85, 88.06) mm, rotated rx 180 ry 0 rz 180 deg; joints [-18.589, 10.738, 64.132, 52.187, 23.798, -49.696]
  Call Extruder(207.86693)
  MoveL 5867 to (239.56, 45.03, 88.06) mm, rotated rx 180 ry 0 rz 180 deg; joints [-18.607, 10.759, 64.108, 52.208, 23.814, -49.715]
  MoveL 5868 to (239.56, 45.03, 88.06) mm, rotated rx 180 ry 0 rz 180 deg; joints [-18.607, 10.759, 64.108, 52.208, 23.814, -49.715]
  Call Extruder(207.97927)
  MoveL 5869 to (239.62, 45.22, 88.06) mm, rotated rx -180 ry 0 rz 180 deg; joints [-18.625, 10.78, 64.083, 52.23, 23.83, -49.734]
  MoveL 5870 to (239.62, 45.22, 88.06) mm, rotated rx -180 ry 0 rz 180 deg; joints [-18.625, 10.78, 64.083, 52.23, 23.83, -49.734]
  Call Extruder(208.09117)
  MoveL 5871 to (239.68, 45.41, 88.06) mm, rotated rx 180 ry 0 rz 180 deg; joints [-18.642, 10.801, 64.058, 52.251, 23.846, -49.752]
  MoveL 5872 to (239.68, 45.41, 88.06) mm, rotated rx 180 ry 0 rz 180 deg; joints [-18.642, 10.801, 64.058, 52.251, 23.846, -49.752]
  Call Extruder(208.21257)
  MoveL 5873 to (239.75, 45.62, 88.06) mm, rotated rx 180 ry 0 rz 180 deg; joints [-18.662, 10.823, 64.031, 52.275, 23.863, -49.772]
  MoveL 5874 to (239.75, 45.62, 88.06) mm, rotated rx 180 ry 0 rz 180 deg; joints [-18.662, 10.823, 64.031, 52.275, 23.863, -49.772]
  Call Extruder(208.34336)
  MoveL 5875 to (239.82, 45.84, 88.06) mm, rotated rx -180 ry 0 rz 180 deg; joints [-18.683, 10.847, 64.002, 52.301, 23.882, -49.795]
  MoveL 5876 to (239.82, 45.84, 88.06) mm, rotated rx -180 ry 0 rz 180 deg; joints [-18.683, 10.847, 64.002, 52.301, 23.882, -49.795]
  Call Extruder(208.47359)
  MoveL 5877 to (239.88, 46.06, 88.06) mm, rotated rx -180 ry 0 rz 180 deg; joints [-18.705, 10.871, 63.974, 52.327, 23.901, -49.817]
  MoveL 5878 to (239.88, 46.06, 88.06) mm, rotated rx -180 ry 0 rz 180 deg; joints [-18.705, 10.871, 63.974, 52.327, 23.901, -49.817]
  Call Extruder(208.60325)
  MoveL 5879 to (239.95, 46.29, 88.06) mm, rotated rx 180 ry 0 rz 180 deg; joints [-18.726, 10.896, 63.945, 52.353, 23.92, -49.839]
  MoveL 5880 to (239.95, 46.29, 88.06) mm, rotated rx 180 ry 0 rz 180 deg; joints [-18.726, 10.896, 63.945, 52.353, 23.92, -49.839]
  Call Extruder(208.73235)
  MoveL 5881 to (240.02, 46.51, 88.06) mm, rotated rx 180 ry 0 rz -180 deg; joints [-18.747, 10.92, 63.917, 52.379, 23.939, -49.861]
  MoveL 5882 to (240.02, 46.51, 88.06) mm, rotated rx 180 ry 0 rz -180 deg; joints [-18.747, 10.92, 63.917, 52.379, 23.939, -49.861]
  Call Extruder(208.84740)
  MoveL 5883 to (240.06, 46.72, 88.06) mm, rotated rx 180 ry 0 rz 180 deg; joints [-18.767, 10.939, 63.894, 52.404, 23.957, -49.883]
  MoveL 5884 to (240.06, 46.72, 88.06) mm, rotated rx 180 ry 0 rz 180 deg; joints [-18.767, 10.939, 63.894, 52.404, 23.957, -49.883]
  Call Extruder(208.96201)
  MoveL 5885 to (240.11, 46.92, 88.06) mm, rotated rx -180 ry 0 rz 180 deg; joints [-18.787, 10.958, 63.871, 52.429, 23.974, -49.905]
  MoveL 5886 to (240.11, 46.92, 88.06) mm, rotated rx -180 ry 0 rz 180 deg; joints [-18.787, 10.958, 63.871, 52.429, 23.974, -49.905]
  Call Extruder(209.07616)
  MoveL 5887 to (240.15, 47.12, 88.06) mm, rotated rx -180 ry 0 rz 180 deg; joints [-18.807, 10.977, 63.848, 52.455, 23.992, -49.927]
  MoveL 5888 to (240.15, 47.12, 88.06) mm, rotated rx -180 ry 0 rz 180 deg; joints [-18.807, 10.977, 63.848, 52.455, 23.992, -49.927]
  Call Extruder(209.18985)
  MoveL 5889 to (240.2, 47.33, 88.06) mm, rotated rx 180 ry 0 rz 180 deg; joints [-18.827, 10.997, 63.825, 52.48, 24.01, -49.949]
  MoveL 5890 to (240.2, 47.33, 88.06) mm, rotated rx 180 ry 0 rz 180 deg; joints [-18.827, 10.997, 63.825, 52.48, 24.01, -49.949]
  Call Extruder(209.31526)
  MoveL 5891 to (240.24, 47.56, 88.06) mm, rotated rx 180 ry 0 rz 180 deg; joints [-18.85, 11.018, 63.8, 52.508, 24.029, -49.973]
  MoveL 5892 to (240.24, 47.56, 88.06) mm, rotated rx 180 ry 0 rz 180 deg; joints [-18.85, 11.018, 63.8, 52.508, 24.029, -49.973]
  Call Extruder(209.45224)
  MoveL 5893 to (240.29, 47.8, 88.06) mm, rotated rx 180 ry 0 rz -180 deg; joints [-18.874, 11.04, 63.773, 52.539, 24.05, -50]
  MoveL 5894 to (240.29, 47.8, 88.06) mm, rotated rx 180 ry 0 rz -180 deg; joints [-18.874, 11.04, 63.773, 52.539, 24.05, -50]
  Call Extruder(209.58861)
  MoveL 5895 to (240.34, 48.05, 88.06) mm, rotated rx -180 ry 0 rz 180 deg; joints [-18.899, 11.063, 63.746, 52.57, 24.072, -50.027]
  MoveL 5896 to (240.34, 48.05, 88.06) mm, rotated rx -180 ry 0 rz 180 deg; joints [-18.899, 11.063, 63.746, 52.57, 24.072, -50.027]
  Call Extruder(209.72437)
  MoveL 5897 to (240.39, 48.3, 88.06) mm, rotated rx -180 ry 0 rz 180 deg; joints [-18.923, 11.086, 63.719, 52.601, 24.093, -50.054]
  MoveL 5898 to (240.39, 48.3, 88.06) mm, rotated rx -180 ry 0 rz 180 deg; joints [-18.923, 11.086, 63.719, 52.601, 24.093, -50.054]
  Call Extruder(209.85951)
  MoveL 5899 to (240.44, 48.55, 88.06) mm, rotated rx 180 ry 0 rz 180 deg; joints [-18.948, 11.109, 63.692, 52.632, 24.115, -50.081]
  MoveL 5900 to (240.44, 48.55, 88.06) mm, rotated rx 180 ry 0 rz 180 deg; joints [-18.948, 11.109, 63.692, 52.632, 24.115, -50.081]
  Call Extruder(209.99405)
  MoveL 5901 to (240.49, 48.8, 88.06) mm, rotated rx 180 ry 0 rz 180 deg; joints [-18.973, 11.132, 63.665, 52.663, 24.136, -50.107]
  MoveL 5902 to (240.49, 48.8, 88.06) mm, rotated rx 180 ry 0 rz 180 deg; joints [-18.973, 11.132, 63.665, 52.663, 24.136, -50.107]
  Call Extruder(210.12798)
  MoveL 5903 to (240.54, 49.05, 88.06) mm, rotated rx 180 ry 0 rz 180 deg; joints [-18.997, 11.154, 63.638, 52.693, 24.158, -50.134]
  MoveL 5904 to (240.54, 49.05, 88.06) mm, rotated rx 180 ry 0 rz 180 deg; joints [-18.997, 11.154, 63.638, 52.693, 24.158, -50.134]
  Call Extruder(210.27584)
  MoveL 5905 to (240.59, 49.33, 88.06) mm, rotated rx -180 ry 0 rz 180 deg; joints [-19.025, 11.179, 63.608, 52.728, 24.182, -50.164]
  MoveL 5906 to (240.59, 49.33, 88.06) mm, rotated rx -180 ry 0 rz 180 deg; joints [-19.025, 11.179, 63.608, 52.728, 24.182, -50.164]
  Call Extruder(210.43759)
  MoveL 5907 to (240.64, 49.63, 88.06) mm, rotated rx -180 ry 0 rz 180 deg; joints [-19.055, 11.205, 63.577, 52.767, 24.208, -50.198]
  MoveL 5908 to (240.64, 49.63, 88.06) mm, rotated rx -180 ry 0 rz 180 deg; joints [-19.055, 11.205, 63.577, 52.767, 24.208, -50.198]
  Call Extruder(210.59860)
  MoveL 5909 to (240.69, 49.94, 88.06) mm, rotated rx -180 ry 0 rz 180 deg; joints [-19.086, 11.231, 63.546, 52.805, 24.235, -50.232]
  MoveL 5910 to (240.69, 49.94, 88.06) mm, rotated rx -180 ry 0 rz 180 deg; joints [-19.086, 11.231, 63.546, 52.805, 24.235, -50.232]
  Call Extruder(210.75889)
  MoveL 5911 to (240.74, 50.24, 88.06) mm, rotated rx -180 ry 0 rz 180 deg; joints [-19.116, 11.257, 63.515, 52.844, 24.261, -50.265]
  MoveL 5912 to (240.74, 50.24, 88.06) mm, rotated rx -180 ry 0 rz 180 deg; joints [-19.116, 11.257, 63.515, 52.844, 24.261, -50.265]
  Call Extruder(210.91845)
  MoveL 5913 to (240.78, 50.55, 88.06) mm, rotated rx 180 ry 0 rz 180 deg; joints [-19.146, 11.283, 63.484, 52.882, 24.288, -50.298]
  MoveL 5914 to (240.78, 50.55, 88.06) mm, rotated rx 180 ry 0 rz 180 deg; joints [-19.146, 11.283, 63.484, 52.882, 24.288, -50.298]
  Call Extruder(211.07728)
  MoveL 5915 to (240.83, 50.86, 88.06) mm, rotated rx 180 ry 0 rz 180 deg; joints [-19.177, 11.309, 63.453, 52.92, 24.314, -50.331]
  MoveL 5916 to (240.83, 50.86, 88.06) mm, rotated rx 180 ry 0 rz 180 deg; joints [-19.177, 11.309, 63.453, 52.92, 24.314, -50.331]
  Call Extruder(211.25596)
  MoveL 5917 to (240.88, 51.2, 88.06) mm, rotated rx 180 ry 0 rz 180 deg; joints [-19.212, 11.337, 63.419, 52.965, 24.344, -50.37]
  MoveL 5918 to (240.88, 51.2, 88.06) mm, rotated rx 180 ry 0 rz 180 deg; joints [-19.212, 11.337, 63.419, 52.965, 24.344, -50.37]
  Call Extruder(211.45440)
  MoveL 5919 to (240.92, 51.59, 88.06) mm, rotated rx -180 ry 0 rz 180 deg; joints [-19.251, 11.368, 63.382, 53.014, 24.378, -50.413]
  MoveL 5920 to (240.92, 51.59, 88.06) mm, rotated rx -180 ry 0 rz 180 deg; joints [-19.251, 11.368, 63.382, 53.014, 24.378, -50.413]
  Call Extruder(211.65197)
  MoveL 5921 to (240.97, 51.98, 88.06) mm, rotated rx -180 ry 0 rz -180 deg; joints [-19.29, 11.399, 63.346, 53.064, 24.412, -50.456]
  MoveL 5922 to (240.97, 51.98, 88.06) mm, rotated rx -180 ry 0 rz -180 deg; joints [-19.29, 11.399, 63.346, 53.064, 24.412, -50.456]
  Call Extruder(211.84868)
  MoveL 5923 to (241.02, 52.36, 88.06) mm, rotated rx -180 ry 0 rz 180 deg; joints [-19.329, 11.429, 63.309, 53.114, 24.446, -50.5]
  MoveL 5924 to (241.02, 52.36, 88.06) mm, rotated rx -180 ry 0 rz 180 deg; joints [-19.329, 11.429, 63.309, 53.114, 24.446, -50.5]
  Call Extruder(212.04452)
  MoveL 5925 to (241.06, 52.75, 88.06) mm, rotated rx -180 ry 0 rz -180 deg; joints [-19.368, 11.46, 63.272, 53.163, 24.479, -50.542]
  MoveL 5926 to (241.06, 52.75, 88.06) mm, rotated rx -180 ry 0 rz -180 deg; joints [-19.368, 11.46, 63.272, 53.163, 24.479, -50.542]
  Call Extruder(212.33996)
  MoveL 5927 to (241.11, 53.34, 88.06) mm, rotated rx 180 ry 0 rz 180 deg; joints [-19.428, 11.503, 63.22, 53.24, 24.531, -50.61]
  MoveL 5928 to (241.11, 53.34, 88.06) mm, rotated rx 180 ry 0 rz 180 deg; joints [-19.428, 11.503, 63.22, 53.24, 24.531, -50.61]
  Call Extruder(212.63406)
  MoveL 5929 to (241.15, 53.93, 88.06) mm, rotated rx 180 ry 0 rz 180 deg; joints [-19.488, 11.546, 63.169, 53.317, 24.583, -50.677]
  MoveL 5930 to (241.15, 53.93, 88.06) mm, rotated rx 180 ry 0 rz 180 deg; joints [-19.488, 11.546, 63.169, 53.317, 24.583, -50.677]
  Call Extruder(212.92684)
  MoveL 5931 to (241.2, 54.52, 88.06) mm, rotated rx 180 ry 0 rz -180 deg; joints [-19.548, 11.59, 63.117, 53.393, 24.634, -50.743]
  MoveL 5932 to (241.2, 54.52, 88.06) mm, rotated rx 180 ry 0 rz -180 deg; joints [-19.548, 11.59, 63.117, 53.393, 24.634, -50.743]
  Call Extruder(213.50029)
  MoveL 5933 to (241.25, 55.68, 88.06) mm, rotated rx 180 ry 0 rz 180 deg; joints [-19.668, 11.667, 63.023, 53.547, 24.736, -50.878]
  MoveL 5934 to (241.25, 55.68, 88.06) mm, rotated rx 180 ry 0 rz 180 deg; joints [-19.668, 11.667, 63.023, 53.547, 24.736, -50.878]
  Call Extruder(214.21412)
  MoveL 5935 to (241.29, 57.14, 88.06) mm, rotated rx 180 ry 0 rz 180 deg; joints [-19.819, 11.763, 62.909, 53.74, 24.865, -51.046]
  Call Extruder(256.27901)
  MoveL 5936 to (241.29, 142.86, 88.06) mm, rotated rx -180 ry 0 rz -180 deg; joints [-28.232, 18.444, 54.481, 61.328, 32.626, -57.004]
  Call Extruder(256.70743)
  MoveL 5937 to (241.27, 143.74, 88.06) mm, rotated rx -180 ry 0 rz -180 deg; joints [-28.313, 18.526, 54.374, 61.374, 32.706, -57.03]
  MoveL 5938 to (241.27, 143.74, 88.06) mm, rotated rx -180 ry 0 rz -180 deg; joints [-28.313, 18.526, 54.374, 61.374, 32.706, -57.03]
  Call Extruder(257.28088)
  MoveL 5939 to (241.22, 144.9, 88.06) mm, rotated rx 180 ry 0 rz 180 deg; joints [-28.421, 18.631, 54.235, 61.437, 32.814, -57.067]
  MoveL 5940 to (241.22, 144.9, 88.06) mm, rotated rx 180 ry 0 rz 180 deg; joints [-28.421, 18.631, 54.235, 61.437, 32.814, -57.067]
  Call Extruder(257.71522)
  MoveL 5941 to (241.18, 145.77, 88.06) mm, rotated rx 180 ry 0 rz 180 deg; joints [-28.503, 18.708, 54.132, 61.485, 32.894, -57.096]
  MoveL 5942 to (241.18, 145.77, 88.06) mm, rotated rx 180 ry 0 rz 180 deg; joints [-28.503, 18.708, 54.132, 61.485, 32.894, -57.096]
  Call Extruder(258.00933)
  MoveL 5943 to (241.13, 146.36, 88.06) mm, rotated rx 180 ry 0 rz 180 deg; joints [-28.559, 18.758, 54.067, 61.519, 32.949, -57.117]
  MoveL 5944 to (241.13, 146.36, 88.06) mm, rotated rx 180 ry 0 rz 180 deg; joints [-28.559, 18.758, 54.067, 61.519, 32.949, -57.117]
  Call Extruder(258.30477)
  MoveL 5945 to (241.09, 146.95, 88.06) mm, rotated rx 180 ry 0 rz 180 deg; joints [-28.615, 18.807, 54.001, 61.553, 33.004, -57.137]
  MoveL 5946 to (241.09, 146.95, 88.06) mm, rotated rx 180 ry 0 rz 180 deg; joints [-28.615, 18.807, 54.001, 61.553, 33.004, -57.137]
  Call Extruder(258.55103)
  MoveL 5947 to (241.04, 147.44, 88.06) mm, rotated rx 180 ry 0 rz 180 deg; joints [-28.662, 18.847, 53.948, 61.582, 33.049, -57.155]
  MoveL 5948 to (241.04, 147.44, 88.06) mm, rotated rx 180 ry 0 rz 180 deg; joints [-28.662, 18.847, 53.948, 61.582, 33.049, -57.155]
  Call Extruder(258.74773)
  MoveL 5949 to (240.99, 147.83, 88.06) mm, rotated rx 180 ry 0 rz 180 deg; joints [-28.7, 18.877, 53.908, 61.606, 33.086, -57.17]
  MoveL 5950 to (240.99, 147.83, 88.06) mm, rotated rx 180 ry 0 rz 180 deg; joints [-28.7, 18.877, 53.908, 61.606, 33.086, -57.17]
  Call Extruder(258.94530)
  MoveL 5951 to (240.95, 148.22, 88.06) mm, rotated rx -180 ry 0 rz -180 deg; joints [-28.737, 18.907, 53.868, 61.629, 33.122, -57.186]
  MoveL 5952 to (240.95, 148.22, 88.06) mm, rotated rx -180 ry 0 rz -180 deg; joints [-28.737, 18.907, 53.868, 61.629, 33.122, -57.186]
  Call Extruder(259.14375)
  MoveL 5953 to (240.9, 148.6, 88.06) mm, rotated rx 180 ry 0 rz 180 deg; joints [-28.774, 18.938, 53.828, 61.653, 33.158, -57.201]
  MoveL 5954 to (240.9, 148.6, 88.06) mm, rotated rx 180 ry 0 rz 180 deg; joints [-28.774, 18.938, 53.828, 61.653, 33.158, -57.201]
  Call Extruder(259.34306)
  MoveL 5955 to (240.86, 148.99, 88.06) mm, rotated rx 180 ry 0 rz 180 deg; joints [-28.812, 18.968, 53.788, 61.677, 33.194, -57.216]
  MoveL 5956 to (240.86, 148.99, 88.06) mm, rotated rx 180 ry 0 rz 180 deg; joints [-28.812, 18.968, 53.788, 61.677, 33.194, -57.216]
  Call Extruder(259.50189)
  MoveL 5957 to (240.81, 149.3, 88.06) mm, rotated rx 180 ry 0 rz 180 deg; joints [-28.842, 18.989, 53.759, 61.697, 33.223, -57.229]
  MoveL 5958 to (240.81, 149.3, 88.06) mm, rotated rx 180 ry 0 rz 180 deg; joints [-28.842, 18.989, 53.759, 61.697, 33.223, -57.229]
  Call Extruder(259.66145)
  MoveL 5959 to (240.76, 149.6, 88.06) mm, rotated rx 180 ry 0 rz 180 deg; joints [-28.872, 19.011, 53.73, 61.717, 33.252, -57.243]
  MoveL 5960 to (240.76, 149.6, 88.06) mm, rotated rx 180 ry 0 rz 180 deg; joints [-28.872, 19.011, 53.73, 61.717, 33.252, -57.243]
  Call Extruder(259.82174)
  MoveL 5961 to (240.71, 149.91, 88.06) mm, rotated rx 180 ry 0 rz 180 deg; joints [-28.902, 19.033, 53.701, 61.737, 33.28, -57.256]
  MoveL 5962 to (240.71, 149.91, 88.06) mm, rotated rx 180 ry 0 rz 180 deg; joints [-28.902, 19.033, 53.701, 61.737, 33.28, -57.256]
  Call Extruder(259.98276)
  MoveL 5963 to (240.66, 150.21, 88.06) mm, rotated rx 180 ry 0 rz 180 deg; joints [-28.932, 19.055, 53.672, 61.757, 33.309, -57.269]
  MoveL 5964 to (240.66, 150.21, 88.06) mm, rotated rx 180 ry 0 rz 180 deg; joints [-28.932, 19.055, 53.672, 61.757, 33.309, -57.269]
  Call Extruder(260.14450)
  MoveL 5965 to (240.61, 150.52, 88.06) mm, rotated rx 180 ry 0 rz 180 deg; joints [-28.962, 19.077, 53.643, 61.777, 33.338, -57.282]
  MoveL 5966 to (240.61, 150.52, 88.06) mm, rotated rx 180 ry 0 rz 180 deg; joints [-28.962, 19.077, 53.643, 61.777, 33.338, -57.282]
  Call Extruder(260.30697)
  MoveL 5967 to (240.57, 150.83, 88.06) mm, rotated rx -180 ry 0 rz 180 deg; joints [-28.993, 19.098, 53.614, 61.797, 33.366, -57.295]
  MoveL 5968 to (240.57, 150.83, 88.06) mm, rotated rx -180 ry 0 rz 180 deg; joints [-28.993, 19.098, 53.614, 61.797, 33.366, -57.295]
  Call Extruder(260.44090)
  MoveL 5969 to (240.52, 151.08, 88.06) mm, rotated rx 180 ry 0 rz 180 deg; joints [-29.017, 19.115, 53.593, 61.814, 33.39, -57.307]
  MoveL 5970 to (240.52, 151.08, 88.06) mm, rotated rx 180 ry 0 rz 180 deg; joints [-29.017, 19.115, 53.593, 61.814, 33.39, -57.307]
  Call Extruder(260.57544)
  MoveL 5971 to (240.47, 151.32, 88.06) mm, rotated rx 180 ry 0 rz 180 deg; joints [-29.043, 19.131, 53.571, 61.832, 33.414, -57.319]
  MoveL 5972 to (240.47, 151.32, 88.06) mm, rotated rx 180 ry 0 rz 180 deg; joints [-29.043, 19.131, 53.571, 61.832, 33.414, -57.319]
  Call Extruder(260.71058)
  MoveL 5973 to (240.42, 151.57, 88.06) mm, rotated rx -180 ry 0 rz 180 deg; joints [-29.067, 19.147, 53.55, 61.849, 33.437, -57.331]
  MoveL 5974 to (240.42, 151.57, 88.06) mm, rotated rx -180 ry 0 rz 180 deg; joints [-29.067, 19.147, 53.55, 61.849, 33.437, -57.331]
  Call Extruder(260.84634)
  MoveL 5975 to (240.37, 151.82, 88.06) mm, rotated rx 180 ry 0 rz 180 deg; joints [-29.092, 19.163, 53.528, 61.866, 33.461, -57.343]
  MoveL 5976 to (240.37, 151.82, 88.06) mm, rotated rx 180 ry 0 rz 180 deg; joints [-29.092, 19.163, 53.528, 61.866, 33.461, -57.343]
  Call Extruder(260.98271)
  MoveL 5977 to (240.32, 152.07, 88.06) mm, rotated rx 180 ry 0 rz 180 deg; joints [-29.117, 19.179, 53.507, 61.884, 33.484, -57.355]
  MoveL 5978 to (240.32, 152.07, 88.06) mm, rotated rx 180 ry 0 rz 180 deg; joints [-29.117, 19.179, 53.507, 61.884, 33.484, -57.355]
  Call Extruder(261.11969)
  MoveL 5979 to (240.27, 152.32, 88.06) mm, rotated rx 180 ry 0 rz 180 deg; joints [-29.142, 19.195, 53.485, 61.901, 33.508, -57.366]
  MoveL 5980 to (240.27, 152.32, 88.06) mm, rotated rx 180 ry 0 rz 180 deg; joints [-29.142, 19.195, 53.485, 61.901, 33.508, -57.366]
  Call Extruder(261.25727)
  MoveL 5981 to (240.22, 152.57, 88.06) mm, rotated rx 180 ry 0 rz 180 deg; joints [-29.167, 19.211, 53.464, 61.918, 33.531, -57.378]
  MoveL 5982 to (240.22, 152.57, 88.06) mm, rotated rx 180 ry 0 rz 180 deg; joints [-29.167, 19.211, 53.464, 61.918, 33.531, -57.378]
  Call Extruder(261.37097)
  MoveL 5983 to (240.17, 152.77, 88.06) mm, rotated rx 180 ry 0 rz 180 deg; joints [-29.188, 19.224, 53.447, 61.932, 33.551, -57.388]
  MoveL 5984 to (240.17, 152.77, 88.06) mm, rotated rx 180 ry 0 rz 180 deg; joints [-29.188, 19.224, 53.447, 61.932, 33.551, -57.388]
  Call Extruder(261.48512)
  MoveL 5985 to (240.13, 152.98, 88.06) mm, rotated rx 180 ry 0 rz 180 deg; joints [-29.209, 19.237, 53.43, 61.947, 33.57, -57.398]
  MoveL 5986 to (240.13, 152.98, 88.06) mm, rotated rx 180 ry 0 rz 180 deg; joints [-29.209, 19.237, 53.43, 61.947, 33.57, -57.398]
  Call Extruder(261.59972)
  MoveL 5987 to (240.08, 153.18, 88.06) mm, rotated rx 180 ry 0 rz -180 deg; joints [-29.229, 19.249, 53.413, 61.961, 33.589, -57.408]
  MoveL 5988 to (240.08, 153.18, 88.06) mm, rotated rx 180 ry 0 rz -180 deg; joints [-29.229, 19.249, 53.413, 61.961, 33.589, -57.408]
  Call Extruder(261.71478)
  MoveL 5989 to (240.04, 153.39, 88.06) mm, rotated rx 180 ry 0 rz 180 deg; joints [-29.25, 19.262, 53.396, 61.976, 33.609, -57.418]
  MoveL 5990 to (240.04, 153.39, 88.06) mm, rotated rx 180 ry 0 rz 180 deg; joints [-29.25, 19.262, 53.396, 61.976, 33.609, -57.418]
  Call Extruder(261.83700)
  MoveL 5991 to (239.98, 153.6, 88.06) mm, rotated rx -180 ry 0 rz 180 deg; joints [-29.272, 19.274, 53.381, 61.992, 33.629, -57.43]
  MoveL 5992 to (239.98, 153.6, 88.06) mm, rotated rx -180 ry 0 rz 180 deg; joints [-29.272, 19.274, 53.381, 61.992, 33.629, -57.43]
  Call Extruder(261.96666)
  MoveL 5993 to (239.92, 153.82, 88.06) mm, rotated rx 180 ry 0 rz -180 deg; joints [-29.296, 19.284, 53.367, 62.01, 33.651, -57.443]
  MoveL 5994 to (239.92, 153.82, 88.06) mm, rotated rx 180 ry 0 rz -180 deg; joints [-29.296, 19.284, 53.367, 62.01, 33.651, -57.443]
  Call Extruder(262.09688)
  MoveL 5995 to (239.85, 154.05, 88.06) mm, rotated rx -180 ry 0 rz 180 deg; joints [-29.319, 19.294, 53.353, 62.029, 33.672, -57.457]
  MoveL 5996 to (239.85, 154.05, 88.06) mm, rotated rx -180 ry 0 rz 180 deg; joints [-29.319, 19.294, 53.353, 62.029, 33.672, -57.457]
  Call Extruder(262.22767)
  MoveL 5997 to (239.78, 154.27, 88.06) mm, rotated rx 180 ry 0 rz 180 deg; joints [-29.343, 19.305, 53.339, 62.047, 33.694, -57.47]
  MoveL 5998 to (239.78, 154.27, 88.06) mm, rotated rx 180 ry 0 rz 180 deg; joints [-29.343, 19.305, 53.339, 62.047, 33.694, -57.47]
  Call Extruder(262.35903)
  MoveL 5999 to (239.71, 154.5, 88.06) mm, rotated rx 180 ry 0 rz 180 deg; joints [-29.366, 19.316, 53.325, 62.065, 33.715, -57.483]
  MoveL 6000 to (239.71, 154.5, 88.06) mm, rotated rx 180 ry 0 rz 180 deg; joints [-29.366, 19.316, 53.325, 62.065, 33.715, -57.483]
  Call Extruder(262.47093)
  MoveL 6001 to (239.65, 154.68, 88.06) mm, rotated rx 180 ry 0 rz 180 deg; joints [-29.386, 19.324, 53.314, 62.081, 33.733, -57.495]
  MoveL 6002 to (239.65, 154.68, 88.06) mm, rotated rx 180 ry 0 rz 180 deg; joints [-29.386, 19.324, 53.314, 62.081, 33.733, -57.495]
  Call Extruder(262.58328)
  MoveL 6003 to (239.59, 154.87, 88.06) mm, rotated rx 180 ry 0 rz 180 deg; joints [-29.406, 19.332, 53.303, 62.096, 33.752, -57.507]
  MoveL 6004 to (239.59, 154.87, 88.06) mm, rotated rx 180 ry 0 rz 180 deg; joints [-29.406, 19.332, 53.303, 62.096, 33.752, -57.507]
  Call Extruder(262.69607)
  MoveL 6005 to (239.53, 155.06, 88.06) mm, rotated rx 180 ry 0 rz 180 deg; joints [-29.426, 19.34, 53.292, 62.112, 33.77, -57.519]
  MoveL 6006 to (239.53, 155.06, 88.06) mm, rotated rx 180 ry 0 rz 180 deg; joints [-29.426, 19.34, 53.292, 62.112, 33.77, -57.519]
  Call Extruder(262.80930)
  MoveL 6007 to (239.47, 155.25, 88.06) mm, rotated rx 180 ry 0 rz 180 deg; joints [-29.446, 19.348, 53.281, 62.128, 33.788, -57.53]
  MoveL 6008 to (239.47, 155.25, 88.06) mm, rotated rx 180 ry 0 rz 180 deg; joints [-29.446, 19.348, 53.281, 62.128, 33.788, -57.53]
  Call Extruder(262.92298)
  MoveL 6009 to (239.41, 155.44, 88.06) mm, rotated rx -180 ry 0 rz 180 deg; joints [-29.466, 19.356, 53.27, 62.143, 33.806, -57.542]
  MoveL 6010 to (239.41, 155.44, 88.06) mm, rotated rx -180 ry 0 rz 180 deg; joints [-29.466, 19.356, 53.27, 62.143, 33.806, -57.542]
  Call Extruder(263.10494)
  MoveL 6011 to (239.29, 155.73, 88.06) mm, rotated rx 180 ry 0 rz 180 deg; joints [-29.499, 19.364, 53.259, 62.171, 33.835, -57.564]
  MoveL 6012 to (239.29, 155.73, 88.06) mm, rotated rx 180 ry 0 rz 180 deg; joints [-29.499, 19.364, 53.259, 62.171, 33.835, -57.564]
  Call Extruder(263.28765)
  MoveL 6013 to (239.16, 156.02, 88.06) mm, rotated rx 180 ry 0 rz 180 deg; joints [-29.531, 19.372, 53.248, 62.199, 33.863, -57.585]
  MoveL 6014 to (239.16, 156.02, 88.06) mm, rotated rx 180 ry 0 rz 180 deg; joints [-29.531, 19.372, 53.248, 62.199, 33.863, -57.585]
  Call Extruder(263.45808)
  MoveL 6015 to (239.05, 156.29, 88.06) mm, rotated rx 180 ry 0 rz -180 deg; joints [-29.561, 19.38, 53.239, 62.224, 33.89, -57.605]
  MoveL 6016 to (239.05, 156.29, 88.06) mm, rotated rx 180 ry 0 rz -180 deg; joints [-29.561, 19.38, 53.239, 62.224, 33.89, -57.605]
  Call Extruder(263.61609)
  MoveL 6017 to (238.94, 156.54, 88.06) mm, rotated rx -180 ry 0 rz 180 deg; joints [-29.589, 19.386, 53.231, 62.248, 33.914, -57.624]
  MoveL 6018 to (238.94, 156.54, 88.06) mm, rotated rx -180 ry 0 rz 180 deg; joints [-29.589, 19.386, 53.231, 62.248, 33.914, -57.624]
  Call Extruder(263.77470)
  MoveL 6019 to (238.84, 156.79, 88.06) mm, rotated rx 180 ry 0 rz 180 deg; joints [-29.617, 19.392, 53.222, 62.272, 33.939, -57.643]
  MoveL 6020 to (238.84, 156.79, 88.06) mm, rotated rx 180 ry 0 rz 180 deg; joints [-29.617, 19.392, 53.222, 62.272, 33.939, -57.643]
  Call Extruder(263.98087)
  MoveL 6021 to (238.66, 157.09, 88.06) mm, rotated rx 180 ry 0 rz 180 deg; joints [-29.653, 19.392, 53.223, 62.307, 33.969, -57.672]
  MoveL 6022 to (238.66, 157.09, 88.06) mm, rotated rx 180 ry 0 rz 180 deg; joints [-29.653, 19.392, 53.223, 62.307, 33.969, -57.672]
  Call Extruder(264.18782)
  MoveL 6023 to (238.49, 157.4, 88.06) mm, rotated rx -180 ry 0 rz 180 deg; joints [-29.689, 19.391, 53.223, 62.342, 34, -57.701]
  MoveL 6024 to (238.49, 157.4, 88.06) mm, rotated rx -180 ry 0 rz 180 deg; joints [-29.689, 19.391, 53.223, 62.342, 34, -57.701]
  Call Extruder(264.39555)
  MoveL 6025 to (238.31, 157.7, 88.06) mm, rotated rx -180 ry 0 rz -180 deg; joints [-29.725, 19.391, 53.224, 62.377, 34.03, -57.73]
  MoveL 6026 to (238.31, 157.7, 88.06) mm, rotated rx -180 ry 0 rz -180 deg; joints [-29.725, 19.391, 53.224, 62.377, 34.03, -57.73]
  Call Extruder(264.60405)
  MoveL 6027 to (238.13, 158.01, 88.06) mm, rotated rx -180 ry 0 rz 180 deg; joints [-29.761, 19.391, 53.224, 62.411, 34.061, -57.758]
  MoveL 6028 to (238.13, 158.01, 88.06) mm, rotated rx -180 ry 0 rz 180 deg; joints [-29.761, 19.391, 53.224, 62.411, 34.061, -57.758]
  Call Extruder(264.78359)
  MoveL 6029 to (237.96, 158.25, 88.06) mm, rotated rx 180 ry 0 rz 180 deg; joints [-29.792, 19.384, 53.233, 62.444, 34.086, -57.786]
  MoveL 6030 to (237.96, 158.25, 88.06) mm, rotated rx 180 ry 0 rz 180 deg; joints [-29.792, 19.384, 53.233, 62.444, 34.086, -57.786]
  Call Extruder(265.11700)
  MoveL 6031 to (237.63, 158.7, 88.06) mm, rotated rx 180 ry 0 rz -180 deg; joints [-29.849, 19.372, 53.25, 62.503, 34.132, -57.838]
  MoveL 6032 to (237.63, 158.7, 88.06) mm, rotated rx 180 ry 0 rz -180 deg; joints [-29.849, 19.372, 53.25, 62.503, 34.132, -57.838]
  Call Extruder(265.45159)
  MoveL 6033 to (237.3, 159.15, 88.06) mm, rotated rx -180 ry 0 rz 180 deg; joints [-29.907, 19.359, 53.266, 62.563, 34.179, -57.889]
  Call Extruder(266.27956)
  MoveL 6034 to (236.39, 160.19, 88.06) mm, rotated rx 180 ry 0 rz 180 deg; joints [-30.046, 19.303, 53.342, 62.72, 34.289, -58.028]
  Call Extruder(267.10747)
  MoveL 6035 to (235.35, 161.1, 88.06) mm, rotated rx 180 ry 0 rz 180 deg; joints [-30.182, 19.211, 53.464, 62.886, 34.389, -58.181]
  Call Extruder(267.27478)
  MoveL 6036 to (235.13, 161.27, 88.06) mm, rotated rx 180 ry 0 rz 180 deg; joints [-30.208, 19.188, 53.495, 62.921, 34.408, -58.214]
  MoveL 6037 to (235.13, 161.27, 88.06) mm, rotated rx 180 ry 0 rz 180 deg; joints [-30.208, 19.188, 53.495, 62.921, 34.408, -58.214]
  Call Extruder(267.60821)
  MoveL 6038 to (234.68, 161.6, 88.06) mm, rotated rx -180 ry 0 rz 180 deg; joints [-30.261, 19.141, 53.557, 62.99, 34.446, -58.279]
  MoveL 6039 to (234.68, 161.6, 88.06) mm, rotated rx -180 ry 0 rz 180 deg; joints [-30.261, 19.141, 53.557, 62.99, 34.446, -58.279]
  Call Extruder(267.94046)
  MoveL 6040 to (234.23, 161.92, 88.06) mm, rotated rx 180 ry 0 rz -180 deg; joints [-30.314, 19.095, 53.619, 63.059, 34.484, -58.343]
  MoveL 6041 to (234.23, 161.92, 88.06) mm, rotated rx 180 ry 0 rz -180 deg; joints [-30.314, 19.095, 53.619, 63.059, 34.484, -58.343]
  Call Extruder(268.05811)
  MoveL 6042 to (234.05, 162.02, 88.06) mm, rotated rx -180 ry 0 rz 180 deg; joints [-30.331, 19.074, 53.646, 63.084, 34.496, -58.368]
  MoveL 6043 to (234.05, 162.02, 88.06) mm, rotated rx -180 ry 0 rz 180 deg; joints [-30.331, 19.074, 53.646, 63.084, 34.496, -58.368]
  Call Extruder(268.26584)
  MoveL 6044 to (233.75, 162.2, 88.06) mm, rotated rx -180 ry 0 rz 180 deg; joints [-30.363, 19.038, 53.694, 63.129, 34.518, -58.41]
  MoveL 6045 to (233.75, 162.2, 88.06) mm, rotated rx -180 ry 0 rz 180 deg; joints [-30.363, 19.038, 53.694, 63.129, 34.518, -58.41]
  Call Extruder(268.47279)
  MoveL 6046 to (233.45, 162.37, 88.06) mm, rotated rx -180 ry 0 rz 180 deg; joints [-30.394, 19.002, 53.742, 63.173, 34.539, -58.453]
  MoveL 6047 to (233.45, 162.37, 88.06) mm, rotated rx -180 ry 0 rz 180 deg; joints [-30.394, 19.002, 53.742, 63.173, 34.539, -58.453]
  Call Extruder(268.67896)
  MoveL 6048 to (233.14, 162.55, 88.06) mm, rotated rx -180 ry 0 rz 180 deg; joints [-30.426, 18.967, 53.79, 63.218, 34.561, -58.496]
  MoveL 6049 to (233.14, 162.55, 88.06) mm, rotated rx -180 ry 0 rz 180 deg; joints [-30.426, 18.967, 53.79, 63.218, 34.561, -58.496]
  Call Extruder(268.86063)
  MoveL 6050 to (232.87, 162.69, 88.06) mm, rotated rx 180 ry 0 rz -180 deg; joints [-30.453, 18.932, 53.835, 63.258, 34.579, -58.534]
  MoveL 6051 to (232.87, 162.69, 88.06) mm, rotated rx 180 ry 0 rz -180 deg; joints [-30.453, 18.932, 53.835, 63.258, 34.579, -58.534]
  Call Extruder(269.01860)
  MoveL 6052 to (232.62, 162.8, 88.06) mm, rotated rx 180 ry 0 rz 180 deg; joints [-30.476, 18.899, 53.879, 63.292, 34.593, -58.568]
  MoveL 6053 to (232.62, 162.8, 88.06) mm, rotated rx 180 ry 0 rz 180 deg; joints [-30.476, 18.899, 53.879, 63.292, 34.593, -58.568]
  Call Extruder(269.17597)
  MoveL 6054 to (232.37, 162.9, 88.06) mm, rotated rx -180 ry 0 rz 180 deg; joints [-30.498, 18.866, 53.923, 63.327, 34.608, -58.602]
  MoveL 6055 to (232.37, 162.9, 88.06) mm, rotated rx -180 ry 0 rz 180 deg; joints [-30.498, 18.866, 53.923, 63.327, 34.608, -58.602]
  Call Extruder(269.35871)
  MoveL 6056 to (232.07, 163.02, 88.06) mm, rotated rx 180 ry 0 rz 180 deg; joints [-30.524, 18.827, 53.975, 63.368, 34.624, -58.642]
  MoveL 6057 to (232.07, 163.02, 88.06) mm, rotated rx 180 ry 0 rz 180 deg; joints [-30.524, 18.827, 53.975, 63.368, 34.624, -58.642]
  Call Extruder(269.54070)
  MoveL 6058 to (231.78, 163.15, 88.06) mm, rotated rx 180 ry 0 rz 180 deg; joints [-30.551, 18.788, 54.027, 63.408, 34.641, -58.682]
  MoveL 6059 to (231.78, 163.15, 88.06) mm, rotated rx 180 ry 0 rz 180 deg; joints [-30.551, 18.788, 54.027, 63.408, 34.641, -58.682]
  Call Extruder(269.68804)
  MoveL 6060 to (231.54, 163.24, 88.06) mm, rotated rx -180 ry 0 rz 180 deg; joints [-30.571, 18.755, 54.071, 63.441, 34.654, -58.715]
  MoveL 6061 to (231.54, 163.24, 88.06) mm, rotated rx -180 ry 0 rz 180 deg; joints [-30.571, 18.755, 54.071, 63.441, 34.654, -58.715]
  Call Extruder(269.80126)
  MoveL 6062 to (231.35, 163.3, 88.06) mm, rotated rx 180 ry 0 rz 180 deg; joints [-30.587, 18.728, 54.107, 63.467, 34.663, -58.74]
  MoveL 6063 to (231.35, 163.3, 88.06) mm, rotated rx 180 ry 0 rz 180 deg; joints [-30.587, 18.728, 54.107, 63.467, 34.663, -58.74]
  Call Extruder(269.91404)
  MoveL 6064 to (231.17, 163.36, 88.06) mm, rotated rx 180 ry 0 rz 180 deg; joints [-30.602, 18.701, 54.142, 63.492, 34.672, -58.765]
  MoveL 6065 to (231.17, 163.36, 88.06) mm, rotated rx 180 ry 0 rz 180 deg; joints [-30.602, 18.701, 54.142, 63.492, 34.672, -58.765]
  Call Extruder(270.02637)
  MoveL 6066 to (230.98, 163.42, 88.06) mm, rotated rx -180 ry 0 rz 180 deg; joints [-30.618, 18.674, 54.178, 63.517, 34.681, -58.791]
  MoveL 6067 to (230.98, 163.42, 88.06) mm, rotated rx -180 ry 0 rz 180 deg; joints [-30.618, 18.674, 54.178, 63.517, 34.681, -58.791]
  Call Extruder(270.13826)
  MoveL 6068 to (230.79, 163.48, 88.06) mm, rotated rx 180 ry 0 rz 180 deg; joints [-30.633, 18.647, 54.214, 63.543, 34.691, -58.816]
  MoveL 6069 to (230.79, 163.48, 88.06) mm, rotated rx 180 ry 0 rz 180 deg; joints [-30.633, 18.647, 54.214, 63.543, 34.691, -58.816]
  Call Extruder(270.25966)
  MoveL 6070 to (230.58, 163.55, 88.06) mm, rotated rx 180 ry 0 rz 180 deg; joints [-30.65, 18.617, 54.253, 63.57, 34.701, -58.843]
  MoveL 6071 to (230.58, 163.55, 88.06) mm, rotated rx 180 ry 0 rz 180 deg; joints [-30.65, 18.617, 54.253, 63.57, 34.701, -58.843]
  Call Extruder(270.39048)
  MoveL 6072 to (230.36, 163.62, 88.06) mm, rotated rx 180 ry 0 rz 180 deg; joints [-30.668, 18.585, 54.296, 63.6, 34.711, -58.873]
  MoveL 6073 to (230.36, 163.62, 88.06) mm, rotated rx 180 ry 0 rz 180 deg; joints [-30.668, 18.585, 54.296, 63.6, 34.711, -58.873]
  Call Extruder(270.52072)
  MoveL 6074 to (230.14, 163.68, 88.06) mm, rotated rx -180 ry 0 rz 180 deg; joints [-30.685, 18.553, 54.338, 63.63, 34.722, -58.903]
  MoveL 6075 to (230.14, 163.68, 88.06) mm, rotated rx -180 ry 0 rz 180 deg; joints [-30.685, 18.553, 54.338, 63.63, 34.722, -58.903]
  Call Extruder(270.65041)
  MoveL 6076 to (229.91, 163.75, 88.06) mm, rotated rx 180 ry 0 rz 180 deg; joints [-30.703, 18.52, 54.381, 63.659, 34.733, -58.933]
  MoveL 6077 to (229.91, 163.75, 88.06) mm, rotated rx 180 ry 0 rz 180 deg; joints [-30.703, 18.52, 54.381, 63.659, 34.733, -58.933]
  Call Extruder(270.77952)
  MoveL 6078 to (229.69, 163.82, 88.06) mm, rotated rx 180 ry 0 rz 180 deg; joints [-30.721, 18.488, 54.424, 63.689, 34.744, -58.962]
  MoveL 6079 to (229.69, 163.82, 88.06) mm, rotated rx 180 ry 0 rz 180 deg; joints [-30.721, 18.488, 54.424, 63.689, 34.744, -58.962]
  Call Extruder(270.89460)
  MoveL 6080 to (229.48, 163.86, 88.06) mm, rotated rx 180 ry 0 rz 180 deg; joints [-30.736, 18.457, 54.465, 63.715, 34.752, -58.989]
  MoveL 6081 to (229.48, 163.86, 88.06) mm, rotated rx 180 ry 0 rz 180 deg; joints [-30.736, 18.457, 54.465, 63.715, 34.752, -58.989]
  Call Extruder(271.00922)
  MoveL 6082 to (229.28, 163.91, 88.06) mm, rotated rx -180 ry 0 rz 180 deg; joints [-30.751, 18.426, 54.506, 63.742, 34.76, -59.016]
  MoveL 6083 to (229.28, 163.91, 88.06) mm, rotated rx -180 ry 0 rz 180 deg; joints [-30.751, 18.426, 54.506, 63.742, 34.76, -59.016]
  Call Extruder(271.12339)
  MoveL 6084 to (229.08, 163.95, 88.06) mm, rotated rx 180 ry 0 rz 180 deg; joints [-30.766, 18.395, 54.547, 63.768, 34.768, -59.042]
  MoveL 6085 to (229.08, 163.95, 88.06) mm, rotated rx 180 ry 0 rz 180 deg; joints [-30.766, 18.395, 54.547, 63.768, 34.768, -59.042]
  Call Extruder(271.23711)
  MoveL 6086 to (228.87, 164, 88.06) mm, rotated rx 180 ry 0 rz 180 deg; joints [-30.781, 18.363, 54.588, 63.794, 34.777, -59.069]
  MoveL 6087 to (228.87, 164, 88.06) mm, rotated rx 180 ry 0 rz 180 deg; joints [-30.781, 18.363, 54.588, 63.794, 34.777, -59.069]
  Call Extruder(271.36253)
  MoveL 6088 to (228.65, 164.04, 88.06) mm, rotated rx -180 ry 0 rz 180 deg; joints [-30.797, 18.329, 54.634, 63.823, 34.786, -59.098]
  MoveL 6089 to (228.65, 164.04, 88.06) mm, rotated rx -180 ry 0 rz 180 deg; joints [-30.797, 18.329, 54.634, 63.823, 34.786, -59.098]
  Call Extruder(271.49950)
  MoveL 6090 to (228.4, 164.09, 88.06) mm, rotated rx 180 ry 0 rz 180 deg; joints [-30.815, 18.29, 54.684, 63.855, 34.796, -59.131]
  MoveL 6091 to (228.4, 164.09, 88.06) mm, rotated rx 180 ry 0 rz 180 deg; joints [-30.815, 18.29, 54.684, 63.855, 34.796, -59.131]
  Call Extruder(271.63587)
  MoveL 6092 to (228.15, 164.14, 88.06) mm, rotated rx -180 ry 0 rz 180 deg; joints [-30.832, 18.252, 54.735, 63.886, 34.806, -59.163]
  MoveL 6093 to (228.15, 164.14, 88.06) mm, rotated rx -180 ry 0 rz 180 deg; joints [-30.832, 18.252, 54.735, 63.886, 34.806, -59.163]
  Call Extruder(271.77163)
  MoveL 6094 to (227.9, 164.19, 88.06) mm, rotated rx 180 ry 0 rz 180 deg; joints [-30.85, 18.214, 54.785, 63.918, 34.816, -59.195]
  MoveL 6095 to (227.9, 164.19, 88.06) mm, rotated rx 180 ry 0 rz 180 deg; joints [-30.85, 18.214, 54.785, 63.918, 34.816, -59.195]
  Call Extruder(271.90678)
  MoveL 6096 to (227.65, 164.24, 88.06) mm, rotated rx -180 ry 0 rz 180 deg; joints [-30.868, 18.175, 54.836, 63.949, 34.825, -59.227]
  MoveL 6097 to (227.65, 164.24, 88.06) mm, rotated rx -180 ry 0 rz 180 deg; joints [-30.868, 18.175, 54.836, 63.949, 34.825, -59.227]
  Call Extruder(272.04131)
  MoveL 6098 to (227.4, 164.29, 88.06) mm, rotated rx 180 ry 0 rz 180 deg; joints [-30.886, 18.137, 54.886, 63.981, 34.835, -59.259]
  MoveL 6099 to (227.4, 164.29, 88.06) mm, rotated rx 180 ry 0 rz 180 deg; joints [-30.886, 18.137, 54.886, 63.981, 34.835, -59.259]
